KUKA KRL program: f1_Kuka_APT226T02S26.SRC

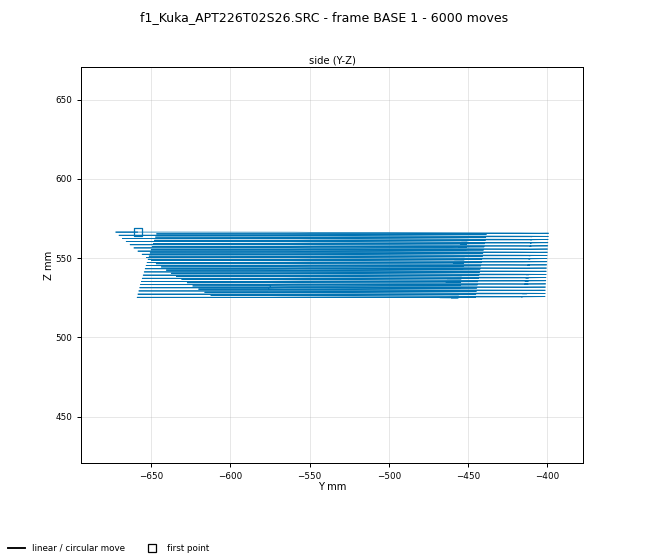
[picture p0: tool path of f1_Kuka_APT226T02S26.SRC in frame BASE 1, 6000 of 6001 moves have a stored position in this frame; points joined in program order, loops and branches not executed]
&ACCESS RVP
&REL 2
&PARAM TEMPLATE = C:\KRC\Roboter\Template\vorgabe
&PARAM EDITMASK = *
DEF f1_Kuka_APT226T02S26()


;FOLD INI;%{PE}%V3.2.0,%MKUKATPBASIS,%CINIT,%VCOMMON,%P
  ;FOLD BAS INI;%{E}%V3.2.0,%MKUKATPBASIS,%CINIT,%VINIT,%P
    GLOBAL INTERRUPT DECL 3 WHEN $STOPMESS==TRUE DO IR_STOPM ( )
    INTERRUPT ON 3
    BAS (#INITMOV,0 )
  ;ENDFOLD (BAS INI)
  ;FOLD USER INI;%{E}%V3.2.0,%MKUKATPUSER,%CINIT,%VINIT,%P
    ;Make your modifications here
  ;ENDFOLD (USER INI)
;ENDFOLD (INI)


;*** Make Null PTP Move
  PTP $pos_act

;*** Auto Load The Correct TOOL Data
  $tool=tool_data[2]

;*** Auto Load The Correct BASE Data
  $base=base_data[1]

  $ADVANCE = 5

;*** Restate Last Velocity
MMPM(30000.0)
SetRPM(8000)
LIN {X 0.091,Y -658.502,Z 566.466,A 0.000,B 0.000,C 90.000,E1 299.922} C_DIS
LIN {X -0.120,Y -661.478,Z 566.462,A 0.000,B 0.000,C 90.000,E1 299.205} C_DIS
LIN {X -0.014,Y -665.940,Z 566.455,A 0.000,B 0.000,C 90.000,E1 297.975} C_DIS
LIN {X 0.167,Y -670.191,Z 566.449,A 0.000,B 0.000,C 90.000,E1 296.744} C_DIS
LIN {X 0.331,Y -670.998,Z 566.447,A 0.000,B 0.000,C 90.000,E1 296.488} C_DIS
LIN {X -0.104,Y -671.526,Z 566.446,A 0.000,B 0.000,C 90.000,E1 296.283} C_DIS
LIN {X -0.059,Y -672.331,Z 566.443,A 0.000,B 0.000,C 90.000,E1 295.796} C_DIS
LIN {X 0.114,Y -672.304,Z 566.442,A 0.000,B 0.000,C 90.000,E1 295.540} C_DIS
LIN {X -0.062,Y -670.081,Z 566.439,A 0.000,B 0.000,C 90.000,E1 294.951} C_DIS
LIN {X 0.021,Y -669.231,Z 566.438,A 0.000,B 0.000,C 90.000,E1 294.823} C_DIS
LIN {X 0.012,Y -665.696,Z 566.436,A 0.000,B 0.000,C 90.000,E1 294.463} C_DIS
LIN {X 0.118,Y -664.657,Z 566.435,A 0.000,B 0.000,C 90.000,E1 294.335} C_DIS
LIN {X 0.191,Y -662.920,Z 566.435,A 0.000,B 0.000,C 90.000,E1 294.207} C_DIS
LIN {X 0.263,Y -660.007,Z 566.434,A 0.000,B 0.000,C 90.000,E1 294.079} C_DIS
LIN {X 0.068,Y -658.610,Z 566.434,A 0.000,B 0.000,C 90.000,E1 294.027} C_DIS
LIN {X -0.130,Y -655.979,Z 566.433,A 0.000,B 0.000,C 90.000,E1 293.875} C_DIS
LIN {X -0.015,Y -649.603,Z 566.431,A 0.000,B 0.000,C 90.000,E1 293.643} C_DIS
LIN {X 0.286,Y -641.955,Z 566.430,A 0.000,B 0.000,C 90.000,E1 293.387} C_DIS
LIN {X -0.348,Y -620.640,Z 566.427,A 0.000,B 0.000,C 90.000,E1 292.898} C_DIS
LIN {X -0.049,Y -600.076,Z 566.424,A 0.000,B 0.000,C 90.000,E1 292.280} C_DIS
LIN {X 0.146,Y -579.548,Z 566.420,A 0.000,B 0.000,C 90.000,E1 291.589} C_DIS
LIN {X 0.178,Y -573.656,Z 566.419,A 0.000,B 0.000,C 90.000,E1 291.354} C_DIS
LIN {X -0.202,Y -567.890,Z 566.417,A 0.000,B 0.000,C 90.000,E1 291.099} C_DIS
LIN {X -0.108,Y -565.511,Z 566.416,A 0.000,B 0.000,C 90.000,E1 290.865} C_DIS
LIN {X 0.054,Y -565.493,Z 566.416,A 0.000,B 0.000,C 90.000,E1 290.844} C_DIS
LIN {X 0.105,Y -565.002,Z 566.415,A 0.000,B 0.000,C 90.000,E1 290.684} C_DIS
LIN {X 0.153,Y -564.693,Z 566.412,A 0.000,B 0.000,C 90.000,E1 290.174} C_DIS
LIN {X 0.335,Y -564.687,Z 566.405,A 0.000,B 0.000,C 90.000,E1 288.779} C_DIS
LIN {X 0.195,Y -564.535,Z 566.398,A 0.000,B 0.000,C 90.000,E1 287.692} C_DIS
LIN {X 0.198,Y -563.994,Z 566.391,A 0.000,B 0.000,C 90.000,E1 286.315} C_DIS
LIN {X 0.039,Y -563.325,Z 566.383,A 0.000,B 0.000,C 90.000,E1 284.954} C_DIS
LIN {X -0.129,Y -562.530,Z 566.375,A 0.000,B 0.000,C 90.000,E1 283.592} C_DIS
LIN {X 0.109,Y -561.743,Z 566.368,A 0.000,B 0.000,C 90.000,E1 282.187} C_DIS
LIN {X -0.215,Y -560.912,Z 566.360,A 0.000,B 0.000,C 90.000,E1 280.838} C_DIS
LIN {X 0.043,Y -559.953,Z 566.351,A 0.000,B 0.000,C 90.000,E1 279.151} C_DIS
LIN {X 0.196,Y -559.248,Z 566.342,A 0.000,B 0.000,C 90.000,E1 277.473} C_DIS
LIN {X -0.153,Y -558.425,Z 566.331,A 0.000,B 0.000,C 90.000,E1 275.568} C_DIS
LIN {X -0.030,Y -557.689,Z 566.320,A 0.000,B 0.000,C 90.000,E1 273.612} C_DIS
LIN {X -0.072,Y -557.116,Z 566.311,A 0.000,B 0.000,C 90.000,E1 271.949} C_DIS
LIN {X -0.206,Y -556.541,Z 566.303,A 0.000,B 0.000,C 90.000,E1 270.573} C_DIS
LIN {X 0.192,Y -555.927,Z 566.295,A 0.000,B 0.000,C 90.000,E1 269.141} C_DIS
LIN {X 0.034,Y -555.274,Z 566.288,A 0.000,B 0.000,C 90.000,E1 267.764} C_DIS
LIN {X -0.133,Y -554.590,Z 566.280,A 0.000,B 0.000,C 90.000,E1 266.388} C_DIS
LIN {X 0.275,Y -553.831,Z 566.272,A 0.000,B 0.000,C 90.000,E1 264.951} C_DIS
LIN {X 0.112,Y -552.989,Z 566.264,A 0.000,B 0.000,C 90.000,E1 263.571} C_DIS
LIN {X -0.049,Y -552.230,Z 566.258,A 0.000,B 0.000,C 90.000,E1 262.470} C_DIS
LIN {X -0.293,Y -551.234,Z 566.252,A 0.000,B 0.000,C 90.000,E1 261.376} C_DIS
LIN {X 0.175,Y -549.737,Z 566.244,A 0.000,B 0.000,C 90.000,E1 259.926} C_DIS
LIN {X -0.258,Y -547.945,Z 566.235,A 0.000,B 0.000,C 90.000,E1 258.285} C_DIS
LIN {X -0.189,Y -546.203,Z 566.225,A 0.000,B 0.000,C 90.000,E1 256.589} C_DIS
LIN {X 0.097,Y -544.289,Z 566.216,A 0.000,B 0.000,C 90.000,E1 254.866} C_DIS
LIN {X 0.116,Y -542.524,Z 566.208,A 0.000,B 0.000,C 90.000,E1 253.449} C_DIS
LIN {X -0.050,Y -540.070,Z 566.199,A 0.000,B 0.000,C 90.000,E1 251.764} C_DIS
LIN {X 0.156,Y -538.266,Z 566.192,A 0.000,B 0.000,C 90.000,E1 250.604} C_DIS
LIN {X -0.135,Y -535.834,Z 566.184,A 0.000,B 0.000,C 90.000,E1 249.209} C_DIS
LIN {X -0.084,Y -532.469,Z 566.175,A 0.000,B 0.000,C 90.000,E1 247.486} C_DIS
LIN {X 0.091,Y -528.786,Z 566.165,A 0.000,B 0.000,C 90.000,E1 245.741} C_DIS
LIN {X 0.230,Y -525.501,Z 566.157,A 0.000,B 0.000,C 90.000,E1 244.280} C_DIS
LIN {X -0.159,Y -521.989,Z 566.149,A 0.000,B 0.000,C 90.000,E1 242.871} C_DIS
LIN {X -0.037,Y -519.122,Z 566.143,A 0.000,B 0.000,C 90.000,E1 241.691} C_DIS
LIN {X 0.046,Y -516.137,Z 566.136,A 0.000,B 0.000,C 90.000,E1 240.511} C_DIS
LIN {X 0.081,Y -512.831,Z 566.130,A 0.000,B 0.000,C 90.000,E1 239.331} C_DIS
LIN {X 0.187,Y -506.734,Z 566.118,A 0.000,B 0.000,C 90.000,E1 237.248} C_DIS
LIN {X -0.020,Y -500.752,Z 566.107,A 0.000,B 0.000,C 90.000,E1 235.182} C_DIS
LIN {X -0.083,Y -493.288,Z 566.092,A 0.000,B 0.000,C 90.000,E1 232.477} C_DIS
LIN {X 0.016,Y -489.998,Z 566.085,A 0.000,B 0.000,C 90.000,E1 231.251} C_DIS
LIN {X -0.175,Y -486.063,Z 566.076,A 0.000,B 0.000,C 90.000,E1 229.747} C_DIS
LIN {X 0.182,Y -480.596,Z 566.064,A 0.000,B 0.000,C 90.000,E1 227.553} C_DIS
LIN {X 0.112,Y -474.437,Z 566.051,A 0.000,B 0.000,C 90.000,E1 225.081} C_DIS
LIN {X -0.068,Y -470.785,Z 566.042,A 0.000,B 0.000,C 90.000,E1 223.542} C_DIS
LIN {X 0.014,Y -467.149,Z 566.033,A 0.000,B 0.000,C 90.000,E1 221.962} C_DIS
LIN {X -0.188,Y -462.845,Z 566.023,A 0.000,B 0.000,C 90.000,E1 220.092} C_DIS
LIN {X -0.252,Y -460.148,Z 566.016,A 0.000,B 0.000,C 90.000,E1 218.830} C_DIS
LIN {X 0.107,Y -455.982,Z 566.005,A 0.000,B 0.000,C 90.000,E1 216.870} C_DIS
LIN {X -0.258,Y -452.625,Z 565.996,A 0.000,B 0.000,C 90.000,E1 215.311} C_DIS
LIN {X -0.238,Y -448.719,Z 565.985,A 0.000,B 0.000,C 90.000,E1 213.372} C_DIS
LIN {X 0.057,Y -444.934,Z 565.974,A 0.000,B 0.000,C 90.000,E1 211.386} C_DIS
LIN {X 0.127,Y -441.936,Z 565.965,A 0.000,B 0.000,C 90.000,E1 209.745} C_DIS
LIN {X 0.041,Y -437.350,Z 565.951,A 0.000,B 0.000,C 90.000,E1 207.129} C_DIS
LIN {X -0.028,Y -433.942,Z 565.940,A 0.000,B 0.000,C 90.000,E1 205.155} C_DIS
LIN {X -0.174,Y -431.214,Z 565.931,A 0.000,B 0.000,C 90.000,E1 203.515} C_DIS
LIN {X 0.020,Y -427.572,Z 565.918,A 0.000,B 0.000,C 90.000,E1 201.153} C_DIS
LIN {X 0.215,Y -425.238,Z 565.908,A 0.000,B 0.000,C 90.000,E1 199.450} C_DIS
LIN {X 0.193,Y -422.028,Z 565.895,A 0.000,B 0.000,C 90.000,E1 197.094} C_DIS
LIN {X -0.161,Y -419.081,Z 565.882,A 0.000,B 0.000,C 90.000,E1 194.773} C_DIS
LIN {X -0.141,Y -417.414,Z 565.874,A 0.000,B 0.000,C 90.000,E1 193.411} C_DIS
LIN {X -0.149,Y -414.490,Z 565.863,A 0.000,B 0.000,C 90.000,E1 191.366} C_DIS
LIN {X -0.153,Y -411.013,Z 565.848,A 0.000,B 0.000,C 90.000,E1 188.624} C_DIS
LIN {X -0.072,Y -408.386,Z 565.834,A 0.000,B 0.000,C 90.000,E1 186.201} C_DIS
LIN {X -0.082,Y -406.582,Z 565.825,A 0.000,B 0.000,C 90.000,E1 184.473} C_DIS
LIN {X 0.071,Y -403.123,Z 565.804,A 0.000,B 0.000,C 90.000,E1 180.630} C_DIS
LIN {X -0.144,Y -401.678,Z 565.792,A 0.000,B 0.000,C 90.000,E1 178.568} C_DIS
LIN {X 0.078,Y -400.698,Z 565.782,A 0.000,B 0.000,C 90.000,E1 176.788} C_DIS
LIN {X 0.151,Y -399.710,Z 565.767,A 0.000,B 0.000,C 90.000,E1 173.976} C_DIS
LIN {X -0.052,Y -399.191,Z 565.749,A 0.000,B 0.000,C 90.000,E1 170.849} C_DIS
LIN {X -0.170,Y -399.159,Z 565.736,A 0.000,B 0.000,C 90.000,E1 168.409} C_DIS
LIN {X 0.025,Y -399.565,Z 565.720,A 0.000,B 0.000,C 90.000,E1 165.574} C_DIS
LIN {X 0.130,Y -399.971,Z 565.712,A 0.000,B 0.000,C 90.000,E1 164.157} C_DIS
LIN {X -0.202,Y -400.926,Z 565.697,A 0.000,B 0.000,C 90.000,E1 161.402} C_DIS
LIN {X 0.084,Y -401.886,Z 565.685,A 0.000,B 0.000,C 90.000,E1 159.263} C_DIS
LIN {X 0.015,Y -402.888,Z 565.673,A 0.000,B 0.000,C 90.000,E1 157.177} C_DIS
LIN {X 0.026,Y -403.897,Z 565.664,A 0.000,B 0.000,C 90.000,E1 155.433} C_DIS
LIN {X 0.112,Y -405.050,Z 565.652,A 0.000,B 0.000,C 90.000,E1 153.332} C_DIS
LIN {X -0.209,Y -406.078,Z 565.642,A 0.000,B 0.000,C 90.000,E1 151.641} C_DIS
LIN {X 0.132,Y -406.794,Z 565.635,A 0.000,B 0.000,C 90.000,E1 150.205} C_DIS
LIN {X 0.039,Y -407.538,Z 565.625,A 0.000,B 0.000,C 90.000,E1 148.486} C_DIS
LIN {X -0.090,Y -408.065,Z 565.617,A 0.000,B 0.000,C 90.000,E1 147.120} C_DIS
LIN {X 0.020,Y -408.430,Z 565.610,A 0.000,B 0.000,C 90.000,E1 145.722} C_DIS
LIN {X 0.053,Y -408.831,Z 565.600,A 0.000,B 0.000,C 90.000,E1 143.989} C_DIS
LIN {X -0.005,Y -409.107,Z 565.590,A 0.000,B 0.000,C 90.000,E1 142.271} C_DIS
LIN {X -0.122,Y -409.308,Z 565.581,A 0.000,B 0.000,C 90.000,E1 140.561} C_DIS
LIN {X -0.083,Y -409.474,Z 565.569,A 0.000,B 0.000,C 90.000,E1 138.485} C_DIS
LIN {X 0.189,Y -409.571,Z 565.558,A 0.000,B 0.000,C 90.000,E1 136.377} C_DIS
LIN {X -0.273,Y -409.836,Z 565.544,A 0.000,B 0.000,C 90.000,E1 134.028} C_DIS
LIN {X -0.141,Y -410.079,Z 565.535,A 0.000,B 0.000,C 90.000,E1 132.285} C_DIS
LIN {X 0.022,Y -410.097,Z 565.525,A 0.000,B 0.000,C 90.000,E1 130.539} C_DIS
LIN {X 0.182,Y -409.998,Z 565.520,A 0.000,B 0.000,C 90.000,E1 129.483} C_DIS
LIN {X 0.080,Y -409.819,Z 565.514,A 0.000,B 0.000,C 90.000,E1 128.463} C_DIS
LIN {X -0.019,Y -409.657,Z 565.511,A 0.000,B 0.000,C 90.000,E1 127.971} C_DIS
LIN {X -0.057,Y -409.666,Z 565.511,A 0.000,B 0.000,C 90.000,E1 127.971} C_DIS
LIN {X -0.188,Y -415.244,Z 565.500,A 0.000,B 0.000,C 90.000,E1 126.091} C_DIS
LIN {X -0.077,Y -416.905,Z 565.497,A 0.000,B 0.000,C 90.000,E1 125.391} C_DIS
LIN {X -0.150,Y -426.632,Z 565.476,A 0.000,B 0.000,C 90.000,E1 121.671} C_DIS
LIN {X -0.187,Y -430.699,Z 565.468,A 0.000,B 0.000,C 90.000,E1 120.335} C_DIS
LIN {X -0.080,Y -437.000,Z 565.454,A 0.000,B 0.000,C 90.000,E1 117.692} C_DIS
LIN {X 0.267,Y -437.037,Z 565.454,A 0.000,B 0.000,C 90.000,E1 117.641} C_DIS
LIN {X -0.240,Y -449.597,Z 565.451,A 0.000,B 0.000,C 90.000,E1 117.129} C_DIS
LIN {X 0.099,Y -461.731,Z 565.448,A 0.000,B 0.000,C 90.000,E1 116.539} C_DIS
LIN {X 0.166,Y -473.663,Z 565.444,A 0.000,B 0.000,C 90.000,E1 115.976} C_DIS
LIN {X -0.213,Y -485.709,Z 565.441,A 0.000,B 0.000,C 90.000,E1 115.463} C_DIS
LIN {X -0.080,Y -495.644,Z 565.439,A 0.000,B 0.000,C 90.000,E1 114.951} C_DIS
LIN {X 0.082,Y -502.219,Z 565.437,A 0.000,B 0.000,C 90.000,E1 114.591} C_DIS
LIN {X 0.151,Y -513.798,Z 565.433,A 0.000,B 0.000,C 90.000,E1 113.951} C_DIS
LIN {X -0.201,Y -525.107,Z 565.430,A 0.000,B 0.000,C 90.000,E1 113.334} C_DIS
LIN {X -0.007,Y -532.885,Z 565.427,A 0.000,B 0.000,C 90.000,E1 112.823} C_DIS
LIN {X 0.033,Y -537.524,Z 565.425,A 0.000,B 0.000,C 90.000,E1 112.514} C_DIS
LIN {X 0.130,Y -546.082,Z 565.422,A 0.000,B 0.000,C 90.000,E1 111.897} C_DIS
LIN {X 0.201,Y -553.885,Z 565.418,A 0.000,B 0.000,C 90.000,E1 111.280} C_DIS
LIN {X 0.052,Y -559.058,Z 565.416,A 0.000,B 0.000,C 90.000,E1 110.844} C_DIS
LIN {X 0.130,Y -563.843,Z 565.413,A 0.000,B 0.000,C 90.000,E1 110.375} C_DIS
LIN {X 0.123,Y -566.067,Z 565.412,A 0.000,B 0.000,C 90.000,E1 110.120} C_DIS
LIN {X 0.206,Y -569.310,Z 565.410,A 0.000,B 0.000,C 90.000,E1 109.758} C_DIS
LIN {X 0.185,Y -573.267,Z 565.407,A 0.000,B 0.000,C 90.000,E1 109.268} C_DIS
LIN {X -0.185,Y -578.969,Z 565.403,A 0.000,B 0.000,C 90.000,E1 108.489} C_DIS
LIN {X -0.093,Y -583.152,Z 565.399,A 0.000,B 0.000,C 90.000,E1 107.819} C_DIS
LIN {X 0.044,Y -589.252,Z 565.393,A 0.000,B 0.000,C 90.000,E1 106.732} C_DIS
LIN {X 0.169,Y -594.082,Z 565.388,A 0.000,B 0.000,C 90.000,E1 105.788} C_DIS
LIN {X 0.006,Y -597.910,Z 565.383,A 0.000,B 0.000,C 90.000,E1 105.009} C_DIS
LIN {X -0.060,Y -600.834,Z 565.380,A 0.000,B 0.000,C 90.000,E1 104.356} C_DIS
LIN {X -0.272,Y -606.577,Z 565.372,A 0.000,B 0.000,C 90.000,E1 103.063} C_DIS
LIN {X -0.133,Y -610.900,Z 565.367,A 0.000,B 0.000,C 90.000,E1 102.007} C_DIS
LIN {X -0.182,Y -615.984,Z 565.359,A 0.000,B 0.000,C 90.000,E1 100.715} C_DIS
LIN {X 0.164,Y -623.736,Z 565.348,A 0.000,B 0.000,C 90.000,E1 98.624} C_DIS
LIN {X -0.289,Y -627.540,Z 565.342,A 0.000,B 0.000,C 90.000,E1 97.644} C_DIS
LIN {X -0.277,Y -632.016,Z 565.335,A 0.000,B 0.000,C 90.000,E1 96.372} C_DIS
LIN {X 0.215,Y -634.479,Z 565.331,A 0.000,B 0.000,C 90.000,E1 95.568} C_DIS
LIN {X 0.108,Y -636.805,Z 565.327,A 0.000,B 0.000,C 90.000,E1 94.821} C_DIS
LIN {X 0.025,Y -638.887,Z 565.323,A 0.000,B 0.000,C 90.000,E1 94.073} C_DIS
LIN {X -0.248,Y -641.332,Z 565.317,A 0.000,B 0.000,C 90.000,E1 93.094} C_DIS
LIN {X 0.081,Y -643.287,Z 565.312,A 0.000,B 0.000,C 90.000,E1 92.064} C_DIS
LIN {X 0.279,Y -644.128,Z 565.309,A 0.000,B 0.000,C 90.000,E1 91.547} C_DIS
LIN {X 0.010,Y -645.490,Z 565.303,A 0.000,B 0.000,C 90.000,E1 90.573} C_DIS
LIN {X -0.016,Y -646.171,Z 565.299,A 0.000,B 0.000,C 90.000,E1 89.828} C_DIS
LIN {X 0.185,Y -646.428,Z 565.296,A 0.000,B 0.000,C 90.000,E1 89.312} C_DIS
LIN {X 0.166,Y -646.585,Z 565.292,A 0.000,B 0.000,C 90.000,E1 88.568} C_DIS
LIN {X 0.166,Y -646.505,Z 565.288,A 0.000,B 0.000,C 90.000,E1 87.822} C_DIS
LIN {X 0.141,Y -646.135,Z 565.284,A 0.000,B 0.000,C 90.000,E1 87.078} C_DIS
LIN {X -0.086,Y -645.321,Z 565.278,A 0.000,B 0.000,C 90.000,E1 86.102} C_DIS
LIN {X -0.273,Y -644.089,Z 565.273,A 0.000,B 0.000,C 90.000,E1 85.122} C_DIS
LIN {X -0.287,Y -643.007,Z 565.269,A 0.000,B 0.000,C 90.000,E1 84.375} C_DIS
LIN {X 0.145,Y -641.255,Z 565.263,A 0.000,B 0.000,C 90.000,E1 83.337} C_DIS
LIN {X -0.350,Y -638.424,Z 565.256,A 0.000,B 0.000,C 90.000,E1 82.129} C_DIS
LIN {X 0.096,Y -635.794,Z 565.251,A 0.000,B 0.000,C 90.000,E1 81.084} C_DIS
LIN {X 0.321,Y -632.160,Z 565.244,A 0.000,B 0.000,C 90.000,E1 79.803} C_DIS
LIN {X -0.135,Y -628.086,Z 565.237,A 0.000,B 0.000,C 90.000,E1 78.578} C_DIS
LIN {X -0.116,Y -625.394,Z 565.232,A 0.000,B 0.000,C 90.000,E1 77.813} C_DIS
LIN {X -0.260,Y -622.564,Z 565.228,A 0.000,B 0.000,C 90.000,E1 77.061} C_DIS
LIN {X 0.228,Y -618.259,Z 565.222,A 0.000,B 0.000,C 90.000,E1 75.992} C_DIS
LIN {X 0.106,Y -614.146,Z 565.217,A 0.000,B 0.000,C 90.000,E1 75.102} C_DIS
LIN {X -0.025,Y -610.337,Z 565.213,A 0.000,B 0.000,C 90.000,E1 74.338} C_DIS
LIN {X 0.010,Y -606.903,Z 565.209,A 0.000,B 0.000,C 90.000,E1 73.685} C_DIS
LIN {X 0.188,Y -603.246,Z 565.206,A 0.000,B 0.000,C 90.000,E1 73.015} C_DIS
LIN {X 0.211,Y -600.152,Z 565.203,A 0.000,B 0.000,C 90.000,E1 72.489} C_DIS
LIN {X -0.232,Y -595.965,Z 565.199,A 0.000,B 0.000,C 90.000,E1 71.873} C_DIS
LIN {X -0.079,Y -592.202,Z 565.196,A 0.000,B 0.000,C 90.000,E1 71.329} C_DIS
LIN {X 0.274,Y -586.514,Z 565.192,A 0.000,B 0.000,C 90.000,E1 70.550} C_DIS
LIN {X -0.192,Y -581.956,Z 565.189,A 0.000,B 0.000,C 90.000,E1 70.061} C_DIS
LIN {X -0.114,Y -577.144,Z 565.186,A 0.000,B 0.000,C 90.000,E1 69.518} C_DIS
LIN {X 0.224,Y -571.989,Z 565.183,A 0.000,B 0.000,C 90.000,E1 68.954} C_DIS
LIN {X -0.098,Y -569.075,Z 565.182,A 0.000,B 0.000,C 90.000,E1 68.720} C_DIS
LIN {X -0.122,Y -567.051,Z 565.181,A 0.000,B 0.000,C 90.000,E1 68.518} C_DIS
LIN {X 0.117,Y -563.879,Z 565.179,A 0.000,B 0.000,C 90.000,E1 68.230} C_DIS
LIN {X 0.190,Y -561.737,Z 565.178,A 0.000,B 0.000,C 90.000,E1 68.028} C_DIS
LIN {X 0.310,Y -555.590,Z 565.175,A 0.000,B 0.000,C 90.000,E1 67.539} C_DIS
LIN {X -0.179,Y -549.616,Z 565.173,A 0.000,B 0.000,C 90.000,E1 67.177} C_DIS
LIN {X 0.018,Y -544.631,Z 565.171,A 0.000,B 0.000,C 90.000,E1 66.847} C_DIS
LIN {X 0.166,Y -538.455,Z 565.169,A 0.000,B 0.000,C 90.000,E1 66.485} C_DIS
LIN {X -0.132,Y -531.737,Z 565.168,A 0.000,B 0.000,C 90.000,E1 66.177} C_DIS
LIN {X -0.018,Y -528.225,Z 565.167,A 0.000,B 0.000,C 90.000,E1 65.997} C_DIS
LIN {X -0.065,Y -516.079,Z 565.164,A 0.000,B 0.000,C 90.000,E1 65.485} C_DIS
LIN {X -0.140,Y -507.333,Z 565.162,A 0.000,B 0.000,C 90.000,E1 65.153} C_DIS
LIN {X -0.033,Y -482.787,Z 565.157,A 0.000,B 0.000,C 90.000,E1 64.229} C_DIS
LIN {X 0.134,Y -463.845,Z 565.153,A 0.000,B 0.000,C 90.000,E1 63.461} C_DIS
LIN {X -0.021,Y -457.694,Z 565.151,A 0.000,B 0.000,C 90.000,E1 63.204} C_DIS
LIN {X -0.056,Y -457.648,Z 565.151,A 0.000,B 0.000,C 90.000,E1 63.204} C_DIS
LIN {X -0.008,Y -455.803,Z 565.145,A 0.000,B 0.000,C 90.000,E1 62.103} C_DIS
LIN {X 0.096,Y -455.205,Z 565.143,A 0.000,B 0.000,C 90.000,E1 61.769} C_DIS
LIN {X -0.056,Y -446.529,Z 565.122,A 0.000,B 0.000,C 90.000,E1 57.916} C_DIS
LIN {X -0.165,Y -444.146,Z 565.115,A 0.000,B 0.000,C 90.000,E1 56.628} C_DIS
LIN {X -0.053,Y -442.565,Z 565.111,A 0.000,B 0.000,C 90.000,E1 55.960} C_DIS
LIN {X 0.165,Y -438.365,Z 565.101,A 0.000,B 0.000,C 90.000,E1 54.196} C_DIS
LIN {X 0.125,Y -438.357,Z 565.101,A 0.000,B 0.000,C 90.000,E1 54.196} C_DIS
LIN {X -0.110,Y -441.521,Z 565.087,A 0.000,B 0.000,C 90.000,E1 51.698} C_DIS
LIN {X -0.174,Y -442.811,Z 565.082,A 0.000,B 0.000,C 90.000,E1 50.723} C_DIS
LIN {X -0.249,Y -445.229,Z 565.071,A 0.000,B 0.000,C 90.000,E1 48.771} C_DIS
LIN {X 0.031,Y -447.166,Z 565.062,A 0.000,B 0.000,C 90.000,E1 47.106} C_DIS
LIN {X 0.000,Y -448.679,Z 565.055,A 0.000,B 0.000,C 90.000,E1 45.810} C_DIS
LIN {X -0.003,Y -449.663,Z 565.049,A 0.000,B 0.000,C 90.000,E1 44.838} C_DIS
LIN {X 0.010,Y -450.802,Z 565.042,A 0.000,B 0.000,C 90.000,E1 43.542} C_DIS
LIN {X 0.058,Y -451.689,Z 565.035,A 0.000,B 0.000,C 90.000,E1 42.243} C_DIS
LIN {X 0.133,Y -452.421,Z 565.026,A 0.000,B 0.000,C 90.000,E1 40.620} C_DIS
LIN {X -0.085,Y -452.674,Z 565.019,A 0.000,B 0.000,C 90.000,E1 39.358} C_DIS
LIN {X -0.016,Y -452.799,Z 565.013,A 0.000,B 0.000,C 90.000,E1 38.382} C_DIS
LIN {X 0.122,Y -452.730,Z 565.006,A 0.000,B 0.000,C 90.000,E1 37.076} C_DIS
LIN {X 0.072,Y -452.492,Z 564.997,A 0.000,B 0.000,C 90.000,E1 35.471} C_DIS
LIN {X 0.074,Y -451.782,Z 564.985,A 0.000,B 0.000,C 90.000,E1 33.214} C_DIS
LIN {X 0.219,Y -451.328,Z 564.974,A 0.000,B 0.000,C 90.000,E1 31.258} C_DIS
LIN {X 0.036,Y -451.029,Z 564.965,A 0.000,B 0.000,C 90.000,E1 29.667} C_DIS
LIN {X 0.191,Y -450.546,Z 564.952,A 0.000,B 0.000,C 90.000,E1 27.385} C_DIS
LIN {X -0.028,Y -450.178,Z 564.943,A 0.000,B 0.000,C 90.000,E1 25.796} C_DIS
LIN {X -0.252,Y -449.954,Z 564.934,A 0.000,B 0.000,C 90.000,E1 24.207} C_DIS
LIN {X 0.094,Y -449.708,Z 564.922,A 0.000,B 0.000,C 90.000,E1 21.897} C_DIS
LIN {X 0.095,Y -449.600,Z 564.909,A 0.000,B 0.000,C 90.000,E1 19.631} C_DIS
LIN {X -0.202,Y -449.669,Z 564.897,A 0.000,B 0.000,C 90.000,E1 17.402} C_DIS
LIN {X 0.107,Y -450.046,Z 564.882,A 0.000,B 0.000,C 90.000,E1 14.773} C_DIS
LIN {X -0.103,Y -450.683,Z 564.870,A 0.000,B 0.000,C 90.000,E1 12.535} C_DIS
LIN {X 0.050,Y -451.603,Z 564.857,A 0.000,B 0.000,C 90.000,E1 10.254} C_DIS
LIN {X 0.175,Y -452.471,Z 564.848,A 0.000,B 0.000,C 90.000,E1 8.624} C_DIS
LIN {X -0.141,Y -454.065,Z 564.834,A 0.000,B 0.000,C 90.000,E1 6.087} C_DIS
LIN {X 0.082,Y -455.571,Z 564.823,A 0.000,B 0.000,C 90.000,E1 4.131} C_DIS
LIN {X -0.219,Y -457.811,Z 564.809,A 0.000,B 0.000,C 90.000,E1 1.604} C_DIS
LIN {X -0.147,Y -460.823,Z 564.794,A 0.000,B 0.000,C 90.000,E1 358.854} C_DIS
LIN {X 0.159,Y -464.118,Z 564.779,A 0.000,B 0.000,C 90.000,E1 356.274} C_DIS
LIN {X 0.159,Y -466.798,Z 564.769,A 0.000,B 0.000,C 90.000,E1 354.375} C_DIS
LIN {X 0.000,Y -469.127,Z 564.760,A 0.000,B 0.000,C 90.000,E1 352.818} C_DIS
LIN {X -0.054,Y -471.385,Z 564.751,A 0.000,B 0.000,C 90.000,E1 351.254} C_DIS
LIN {X -0.238,Y -474.139,Z 564.741,A 0.000,B 0.000,C 90.000,E1 349.398} C_DIS
LIN {X -0.026,Y -476.585,Z 564.732,A 0.000,B 0.000,C 90.000,E1 347.813} C_DIS
LIN {X -0.094,Y -480.574,Z 564.719,A 0.000,B 0.000,C 90.000,E1 345.338} C_DIS
LIN {X 0.067,Y -485.614,Z 564.703,A 0.000,B 0.000,C 90.000,E1 342.543} C_DIS
LIN {X -0.163,Y -489.177,Z 564.693,A 0.000,B 0.000,C 90.000,E1 340.732} C_DIS
LIN {X -0.188,Y -492.149,Z 564.684,A 0.000,B 0.000,C 90.000,E1 339.209} C_DIS
LIN {X -0.027,Y -494.423,Z 564.678,A 0.000,B 0.000,C 90.000,E1 337.975} C_DIS
LIN {X -0.236,Y -497.287,Z 564.669,A 0.000,B 0.000,C 90.000,E1 336.485} C_DIS
LIN {X -0.192,Y -499.962,Z 564.661,A 0.000,B 0.000,C 90.000,E1 334.973} C_DIS
LIN {X -0.104,Y -502.524,Z 564.653,A 0.000,B 0.000,C 90.000,E1 333.461} C_DIS
LIN {X 0.179,Y -504.561,Z 564.646,A 0.000,B 0.000,C 90.000,E1 332.231} C_DIS
LIN {X -0.002,Y -507.496,Z 564.636,A 0.000,B 0.000,C 90.000,E1 330.461} C_DIS
LIN {X 0.108,Y -511.464,Z 564.623,A 0.000,B 0.000,C 90.000,E1 328.074} C_DIS
LIN {X 0.170,Y -514.489,Z 564.613,A 0.000,B 0.000,C 90.000,E1 326.294} C_DIS
LIN {X -0.064,Y -517.057,Z 564.605,A 0.000,B 0.000,C 90.000,E1 324.848} C_DIS
LIN {X 0.041,Y -519.683,Z 564.597,A 0.000,B 0.000,C 90.000,E1 323.371} C_DIS
LIN {X -0.045,Y -523.919,Z 564.584,A 0.000,B 0.000,C 90.000,E1 321.045} C_DIS
LIN {X -0.047,Y -528.029,Z 564.572,A 0.000,B 0.000,C 90.000,E1 319.013} C_DIS
LIN {X -0.004,Y -533.253,Z 564.560,A 0.000,B 0.000,C 90.000,E1 316.701} C_DIS
LIN {X -0.177,Y -537.393,Z 564.550,A 0.000,B 0.000,C 90.000,E1 315.000} C_DIS
LIN {X -0.213,Y -538.687,Z 564.547,A 0.000,B 0.000,C 90.000,E1 314.433} C_DIS
LIN {X 0.115,Y -542.821,Z 564.539,A 0.000,B 0.000,C 90.000,E1 312.975} C_DIS
LIN {X -0.161,Y -545.204,Z 564.535,A 0.000,B 0.000,C 90.000,E1 312.366} C_DIS
LIN {X -0.039,Y -547.320,Z 564.533,A 0.000,B 0.000,C 90.000,E1 312.000} C_DIS
LIN {X 0.160,Y -548.035,Z 564.533,A 0.000,B 0.000,C 90.000,E1 311.838} C_DIS
LIN {X -0.214,Y -550.099,Z 564.531,A 0.000,B 0.000,C 90.000,E1 311.595} C_DIS
LIN {X -0.011,Y -550.977,Z 564.530,A 0.000,B 0.000,C 90.000,E1 311.434} C_DIS
LIN {X -0.171,Y -552.096,Z 564.529,A 0.000,B 0.000,C 90.000,E1 311.310} C_DIS
LIN {X 0.012,Y -553.582,Z 564.529,A 0.000,B 0.000,C 90.000,E1 311.148} C_DIS
LIN {X -0.157,Y -555.670,Z 564.527,A 0.000,B 0.000,C 90.000,E1 310.906} C_DIS
LIN {X 0.040,Y -560.191,Z 564.525,A 0.000,B 0.000,C 90.000,E1 310.458} C_DIS
LIN {X -0.289,Y -566.071,Z 564.522,A 0.000,B 0.000,C 90.000,E1 310.011} C_DIS
LIN {X -0.235,Y -576.106,Z 564.518,A 0.000,B 0.000,C 90.000,E1 309.277} C_DIS
LIN {X -0.055,Y -586.453,Z 564.514,A 0.000,B 0.000,C 90.000,E1 308.508} C_DIS
LIN {X -0.329,Y -592.161,Z 564.512,A 0.000,B 0.000,C 90.000,E1 308.096} C_DIS
LIN {X -0.321,Y -598.973,Z 564.508,A 0.000,B 0.000,C 90.000,E1 307.523} C_DIS
LIN {X -0.155,Y -604.172,Z 564.506,A 0.000,B 0.000,C 90.000,E1 307.030} C_DIS
LIN {X -0.165,Y -607.955,Z 564.504,A 0.000,B 0.000,C 90.000,E1 306.664} C_DIS
LIN {X 0.052,Y -612.817,Z 564.501,A 0.000,B 0.000,C 90.000,E1 306.137} C_DIS
LIN {X -0.272,Y -619.839,Z 564.497,A 0.000,B 0.000,C 90.000,E1 305.391} C_DIS
LIN {X 0.174,Y -628.577,Z 564.491,A 0.000,B 0.000,C 90.000,E1 304.326} C_DIS
LIN {X 0.013,Y -634.783,Z 564.487,A 0.000,B 0.000,C 90.000,E1 303.579} C_DIS
LIN {X -0.102,Y -639.721,Z 564.483,A 0.000,B 0.000,C 90.000,E1 302.959} C_DIS
LIN {X -0.182,Y -643.971,Z 564.480,A 0.000,B 0.000,C 90.000,E1 302.339} C_DIS
LIN {X 0.285,Y -647.097,Z 564.477,A 0.000,B 0.000,C 90.000,E1 301.799} C_DIS
LIN {X -0.074,Y -650.468,Z 564.473,A 0.000,B 0.000,C 90.000,E1 301.209} C_DIS
LIN {X 0.025,Y -654.513,Z 564.469,A 0.000,B 0.000,C 90.000,E1 300.335} C_DIS
LIN {X 0.220,Y -658.730,Z 564.463,A 0.000,B 0.000,C 90.000,E1 299.333} C_DIS
LIN {X 0.279,Y -663.216,Z 564.456,A 0.000,B 0.000,C 90.000,E1 298.103} C_DIS
LIN {X -0.177,Y -667.563,Z 564.450,A 0.000,B 0.000,C 90.000,E1 296.924} C_DIS
LIN {X 0.132,Y -669.149,Z 564.447,A 0.000,B 0.000,C 90.000,E1 296.411} C_DIS
LIN {X 0.160,Y -670.059,Z 564.444,A 0.000,B 0.000,C 90.000,E1 295.924} C_DIS
LIN {X -0.279,Y -670.256,Z 564.443,A 0.000,B 0.000,C 90.000,E1 295.720} C_DIS
LIN {X -0.114,Y -669.973,Z 564.441,A 0.000,B 0.000,C 90.000,E1 295.463} C_DIS
LIN {X 0.052,Y -669.123,Z 564.440,A 0.000,B 0.000,C 90.000,E1 295.207} C_DIS
LIN {X 0.215,Y -668.096,Z 564.439,A 0.000,B 0.000,C 90.000,E1 294.951} C_DIS
LIN {X 0.014,Y -667.068,Z 564.438,A 0.000,B 0.000,C 90.000,E1 294.847} C_DIS
LIN {X 0.096,Y -665.847,Z 564.437,A 0.000,B 0.000,C 90.000,E1 294.719} C_DIS
LIN {X -0.295,Y -664.134,Z 564.436,A 0.000,B 0.000,C 90.000,E1 294.515} C_DIS
LIN {X -0.223,Y -662.944,Z 564.435,A 0.000,B 0.000,C 90.000,E1 294.387} C_DIS
LIN {X -0.150,Y -660.945,Z 564.435,A 0.000,B 0.000,C 90.000,E1 294.259} C_DIS
LIN {X -0.004,Y -659.139,Z 564.434,A 0.000,B 0.000,C 90.000,E1 294.155} C_DIS
LIN {X 0.146,Y -656.365,Z 564.433,A 0.000,B 0.000,C 90.000,E1 293.951} C_DIS
LIN {X -0.119,Y -654.664,Z 564.433,A 0.000,B 0.000,C 90.000,E1 293.875} C_DIS
LIN {X -0.096,Y -649.752,Z 564.432,A 0.000,B 0.000,C 90.000,E1 293.695} C_DIS
LIN {X 0.221,Y -640.602,Z 564.430,A 0.000,B 0.000,C 90.000,E1 293.387} C_DIS
LIN {X 0.091,Y -621.538,Z 564.427,A 0.000,B 0.000,C 90.000,E1 292.898} C_DIS
LIN {X -0.170,Y -601.106,Z 564.424,A 0.000,B 0.000,C 90.000,E1 292.333} C_DIS
LIN {X -0.148,Y -580.528,Z 564.420,A 0.000,B 0.000,C 90.000,E1 291.663} C_DIS
LIN {X 0.043,Y -573.386,Z 564.419,A 0.000,B 0.000,C 90.000,E1 291.354} C_DIS
LIN {X 0.224,Y -568.086,Z 564.417,A 0.000,B 0.000,C 90.000,E1 291.046} C_DIS
LIN {X 0.017,Y -566.082,Z 564.416,A 0.000,B 0.000,C 90.000,E1 290.865} C_DIS
LIN {X -0.024,Y -566.046,Z 564.416,A 0.000,B 0.000,C 90.000,E1 290.865} C_DIS
LIN {X 0.193,Y -565.520,Z 564.415,A 0.000,B 0.000,C 90.000,E1 290.663} C_DIS
LIN {X -0.203,Y -565.309,Z 564.413,A 0.000,B 0.000,C 90.000,E1 290.429} C_DIS
LIN {X -0.066,Y -565.165,Z 564.403,A 0.000,B 0.000,C 90.000,E1 288.489} C_DIS
LIN {X -0.194,Y -564.948,Z 564.397,A 0.000,B 0.000,C 90.000,E1 287.402} C_DIS
LIN {X -0.177,Y -564.356,Z 564.389,A 0.000,B 0.000,C 90.000,E1 286.024} C_DIS
LIN {X -0.181,Y -563.658,Z 564.381,A 0.000,B 0.000,C 90.000,E1 284.647} C_DIS
LIN {X 0.066,Y -562.845,Z 564.374,A 0.000,B 0.000,C 90.000,E1 283.244} C_DIS
LIN {X 0.275,Y -562.214,Z 564.368,A 0.000,B 0.000,C 90.000,E1 282.119} C_DIS
LIN {X -0.157,Y -561.407,Z 564.360,A 0.000,B 0.000,C 90.000,E1 280.782} C_DIS
LIN {X 0.114,Y -560.465,Z 564.351,A 0.000,B 0.000,C 90.000,E1 279.095} C_DIS
LIN {X -0.201,Y -559.791,Z 564.341,A 0.000,B 0.000,C 90.000,E1 277.466} C_DIS
LIN {X -0.054,Y -558.936,Z 564.331,A 0.000,B 0.000,C 90.000,E1 275.511} C_DIS
LIN {X 0.084,Y -558.205,Z 564.320,A 0.000,B 0.000,C 90.000,E1 273.555} C_DIS
LIN {X 0.054,Y -557.602,Z 564.311,A 0.000,B 0.000,C 90.000,E1 271.892} C_DIS
LIN {X -0.073,Y -557.024,Z 564.303,A 0.000,B 0.000,C 90.000,E1 270.516} C_DIS
LIN {X -0.223,Y -556.402,Z 564.295,A 0.000,B 0.000,C 90.000,E1 269.141} C_DIS
LIN {X 0.260,Y -555.547,Z 564.286,A 0.000,B 0.000,C 90.000,E1 267.421} C_DIS
LIN {X 0.023,Y -555.000,Z 564.280,A 0.000,B 0.000,C 90.000,E1 266.331} C_DIS
LIN {X -0.224,Y -554.397,Z 564.273,A 0.000,B 0.000,C 90.000,E1 265.241} C_DIS
LIN {X -0.270,Y -553.367,Z 564.264,A 0.000,B 0.000,C 90.000,E1 263.571} C_DIS
LIN {X 0.164,Y -552.396,Z 564.256,A 0.000,B 0.000,C 90.000,E1 262.129} C_DIS
LIN {X -0.118,Y -551.618,Z 564.252,A 0.000,B 0.000,C 90.000,E1 261.319} C_DIS
LIN {X -0.187,Y -550.118,Z 564.244,A 0.000,B 0.000,C 90.000,E1 259.926} C_DIS
LIN {X -0.181,Y -548.577,Z 564.236,A 0.000,B 0.000,C 90.000,E1 258.522} C_DIS
LIN {X -0.100,Y -546.858,Z 564.227,A 0.000,B 0.000,C 90.000,E1 256.825} C_DIS
LIN {X 0.199,Y -544.907,Z 564.217,A 0.000,B 0.000,C 90.000,E1 255.102} C_DIS
LIN {X -0.060,Y -542.797,Z 564.208,A 0.000,B 0.000,C 90.000,E1 253.433} C_DIS
LIN {X 0.139,Y -540.271,Z 564.199,A 0.000,B 0.000,C 90.000,E1 251.710} C_DIS
LIN {X 0.123,Y -538.899,Z 564.194,A 0.000,B 0.000,C 90.000,E1 250.859} C_DIS
LIN {X 0.026,Y -536.476,Z 564.186,A 0.000,B 0.000,C 90.000,E1 249.444} C_DIS
LIN {X -0.026,Y -534.844,Z 564.181,A 0.000,B 0.000,C 90.000,E1 248.592} C_DIS
LIN {X 0.096,Y -532.588,Z 564.175,A 0.000,B 0.000,C 90.000,E1 247.433} C_DIS
LIN {X 0.082,Y -529.484,Z 564.167,A 0.000,B 0.000,C 90.000,E1 245.997} C_DIS
LIN {X -0.074,Y -525.552,Z 564.157,A 0.000,B 0.000,C 90.000,E1 244.280} C_DIS
LIN {X 0.005,Y -521.984,Z 564.149,A 0.000,B 0.000,C 90.000,E1 242.820} C_DIS
LIN {X -0.208,Y -518.373,Z 564.141,A 0.000,B 0.000,C 90.000,E1 241.385} C_DIS
LIN {X 0.198,Y -516.122,Z 564.136,A 0.000,B 0.000,C 90.000,E1 240.461} C_DIS
LIN {X -0.127,Y -513.684,Z 564.131,A 0.000,B 0.000,C 90.000,E1 239.616} C_DIS
LIN {X -0.066,Y -508.391,Z 564.121,A 0.000,B 0.000,C 90.000,E1 237.837} C_DIS
LIN {X 0.313,Y -503.196,Z 564.111,A 0.000,B 0.000,C 90.000,E1 236.008} C_DIS
LIN {X -0.143,Y -498.940,Z 564.103,A 0.000,B 0.000,C 90.000,E1 234.562} C_DIS
LIN {X 0.017,Y -493.169,Z 564.091,A 0.000,B 0.000,C 90.000,E1 232.431} C_DIS
LIN {X 0.242,Y -487.522,Z 564.080,A 0.000,B 0.000,C 90.000,E1 230.275} C_DIS
LIN {X -0.177,Y -482.779,Z 564.069,A 0.000,B 0.000,C 90.000,E1 228.485} C_DIS
LIN {X -0.109,Y -480.476,Z 564.064,A 0.000,B 0.000,C 90.000,E1 227.553} C_DIS
LIN {X -0.179,Y -474.317,Z 564.050,A 0.000,B 0.000,C 90.000,E1 225.081} C_DIS
LIN {X -0.018,Y -470.670,Z 564.042,A 0.000,B 0.000,C 90.000,E1 223.500} C_DIS
LIN {X 0.071,Y -467.013,Z 564.033,A 0.000,B 0.000,C 90.000,E1 221.919} C_DIS
LIN {X 0.122,Y -463.448,Z 564.024,A 0.000,B 0.000,C 90.000,E1 220.334} C_DIS
LIN {X 0.103,Y -460.005,Z 564.015,A 0.000,B 0.000,C 90.000,E1 218.749} C_DIS
LIN {X -0.184,Y -455.842,Z 564.005,A 0.000,B 0.000,C 90.000,E1 216.870} C_DIS
LIN {X 0.168,Y -451.824,Z 563.994,A 0.000,B 0.000,C 90.000,E1 214.898} C_DIS
LIN {X -0.134,Y -447.256,Z 563.981,A 0.000,B 0.000,C 90.000,E1 212.673} C_DIS
LIN {X 0.143,Y -444.766,Z 563.974,A 0.000,B 0.000,C 90.000,E1 211.337} C_DIS
LIN {X -0.118,Y -441.186,Z 563.963,A 0.000,B 0.000,C 90.000,E1 209.411} C_DIS
LIN {X 0.133,Y -437.175,Z 563.951,A 0.000,B 0.000,C 90.000,E1 207.078} C_DIS
LIN {X 0.065,Y -433.780,Z 563.940,A 0.000,B 0.000,C 90.000,E1 205.103} C_DIS
LIN {X -0.079,Y -431.048,Z 563.930,A 0.000,B 0.000,C 90.000,E1 203.462} C_DIS
LIN {X -0.087,Y -427.942,Z 563.919,A 0.000,B 0.000,C 90.000,E1 201.461} C_DIS
LIN {X -0.088,Y -425.088,Z 563.908,A 0.000,B 0.000,C 90.000,E1 199.450} C_DIS
LIN {X 0.111,Y -422.376,Z 563.897,A 0.000,B 0.000,C 90.000,E1 197.402} C_DIS
LIN {X -0.060,Y -418.993,Z 563.882,A 0.000,B 0.000,C 90.000,E1 194.717} C_DIS
LIN {X -0.095,Y -417.803,Z 563.876,A 0.000,B 0.000,C 90.000,E1 193.703} C_DIS
LIN {X 0.159,Y -416.324,Z 563.870,A 0.000,B 0.000,C 90.000,E1 192.647} C_DIS
LIN {X -0.158,Y -412.215,Z 563.853,A 0.000,B 0.000,C 90.000,E1 189.613} C_DIS
LIN {X 0.056,Y -408.721,Z 563.836,A 0.000,B 0.000,C 90.000,E1 186.486} C_DIS
LIN {X 0.021,Y -406.566,Z 563.825,A 0.000,B 0.000,C 90.000,E1 184.416} C_DIS
LIN {X -0.196,Y -403.423,Z 563.805,A 0.000,B 0.000,C 90.000,E1 180.974} C_DIS
LIN {X -0.040,Y -401.710,Z 563.792,A 0.000,B 0.000,C 90.000,E1 178.511} C_DIS
LIN {X 0.012,Y -400.178,Z 563.774,A 0.000,B 0.000,C 90.000,E1 175.355} C_DIS
LIN {X -0.177,Y -399.634,Z 563.763,A 0.000,B 0.000,C 90.000,E1 173.280} C_DIS
LIN {X 0.022,Y -399.294,Z 563.745,A 0.000,B 0.000,C 90.000,E1 170.095} C_DIS
LIN {X -0.041,Y -399.406,Z 563.729,A 0.000,B 0.000,C 90.000,E1 167.297} C_DIS
LIN {X -0.149,Y -400.129,Z 563.712,A 0.000,B 0.000,C 90.000,E1 164.157} C_DIS
LIN {X 0.032,Y -401.095,Z 563.696,A 0.000,B 0.000,C 90.000,E1 161.329} C_DIS
LIN {X 0.189,Y -402.052,Z 563.685,A 0.000,B 0.000,C 90.000,E1 159.209} C_DIS
LIN {X 0.079,Y -403.491,Z 563.669,A 0.000,B 0.000,C 90.000,E1 156.433} C_DIS
LIN {X -0.098,Y -404.481,Z 563.659,A 0.000,B 0.000,C 90.000,E1 154.717} C_DIS
LIN {X 0.177,Y -406.125,Z 563.644,A 0.000,B 0.000,C 90.000,E1 151.897} C_DIS
LIN {X -0.122,Y -407.037,Z 563.634,A 0.000,B 0.000,C 90.000,E1 150.205} C_DIS
LIN {X 0.003,Y -407.765,Z 563.625,A 0.000,B 0.000,C 90.000,E1 148.456} C_DIS
LIN {X 0.143,Y -408.378,Z 563.615,A 0.000,B 0.000,C 90.000,E1 146.707} C_DIS
LIN {X 0.114,Y -408.674,Z 563.609,A 0.000,B 0.000,C 90.000,E1 145.674} C_DIS
LIN {X -0.186,Y -409.091,Z 563.600,A 0.000,B 0.000,C 90.000,E1 143.989} C_DIS
LIN {X -0.238,Y -409.364,Z 563.590,A 0.000,B 0.000,C 90.000,E1 142.271} C_DIS
LIN {X -0.035,Y -409.527,Z 563.581,A 0.000,B 0.000,C 90.000,E1 140.517} C_DIS
LIN {X 0.119,Y -409.671,Z 563.571,A 0.000,B 0.000,C 90.000,E1 138.771} C_DIS
LIN {X 0.121,Y -409.747,Z 563.560,A 0.000,B 0.000,C 90.000,E1 136.701} C_DIS
LIN {X 0.242,Y -409.987,Z 563.546,A 0.000,B 0.000,C 90.000,E1 134.271} C_DIS
LIN {X -0.201,Y -410.236,Z 563.537,A 0.000,B 0.000,C 90.000,E1 132.609} C_DIS
LIN {X -0.030,Y -410.301,Z 563.527,A 0.000,B 0.000,C 90.000,E1 130.862} C_DIS
LIN {X 0.136,Y -410.286,Z 563.521,A 0.000,B 0.000,C 90.000,E1 129.806} C_DIS
LIN {X -0.119,Y -410.000,Z 563.514,A 0.000,B 0.000,C 90.000,E1 128.463} C_DIS
LIN {X -0.119,Y -409.793,Z 563.511,A 0.000,B 0.000,C 90.000,E1 127.935} C_DIS
LIN {X 0.165,Y -409.803,Z 563.511,A 0.000,B 0.000,C 90.000,E1 127.890} C_DIS
LIN {X 0.195,Y -415.328,Z 563.500,A 0.000,B 0.000,C 90.000,E1 126.011} C_DIS
LIN {X -0.148,Y -418.583,Z 563.493,A 0.000,B 0.000,C 90.000,E1 124.692} C_DIS
LIN {X 0.212,Y -428.712,Z 563.472,A 0.000,B 0.000,C 90.000,E1 120.924} C_DIS
LIN {X 0.202,Y -430.773,Z 563.468,A 0.000,B 0.000,C 90.000,E1 120.256} C_DIS
LIN {X 0.129,Y -437.732,Z 563.452,A 0.000,B 0.000,C 90.000,E1 117.385} C_DIS
LIN {X 0.089,Y -437.794,Z 563.452,A 0.000,B 0.000,C 90.000,E1 117.385} C_DIS
LIN {X -0.120,Y -460.944,Z 563.446,A 0.000,B 0.000,C 90.000,E1 116.360} C_DIS
LIN {X -0.021,Y -472.889,Z 563.443,A 0.000,B 0.000,C 90.000,E1 115.796} C_DIS
LIN {X 0.291,Y -484.997,Z 563.440,A 0.000,B 0.000,C 90.000,E1 115.207} C_DIS
LIN {X -0.163,Y -494.941,Z 563.438,A 0.000,B 0.000,C 90.000,E1 114.771} C_DIS
LIN {X 0.220,Y -501.677,Z 563.436,A 0.000,B 0.000,C 90.000,E1 114.387} C_DIS
LIN {X 0.040,Y -514.814,Z 563.432,A 0.000,B 0.000,C 90.000,E1 113.695} C_DIS
LIN {X 0.098,Y -524.575,Z 563.429,A 0.000,B 0.000,C 90.000,E1 113.131} C_DIS
LIN {X 0.165,Y -532.372,Z 563.426,A 0.000,B 0.000,C 90.000,E1 112.642} C_DIS
LIN {X -0.113,Y -538.331,Z 563.424,A 0.000,B 0.000,C 90.000,E1 112.280} C_DIS
LIN {X -0.132,Y -541.470,Z 563.423,A 0.000,B 0.000,C 90.000,E1 112.078} C_DIS
LIN {X -0.081,Y -547.464,Z 563.420,A 0.000,B 0.000,C 90.000,E1 111.642} C_DIS
LIN {X 0.081,Y -552.739,Z 563.418,A 0.000,B 0.000,C 90.000,E1 111.227} C_DIS
LIN {X -0.018,Y -558.046,Z 563.416,A 0.000,B 0.000,C 90.000,E1 110.791} C_DIS
LIN {X -0.008,Y -563.246,Z 563.413,A 0.000,B 0.000,C 90.000,E1 110.301} C_DIS
LIN {X 0.100,Y -568.271,Z 563.410,A 0.000,B 0.000,C 90.000,E1 109.758} C_DIS
LIN {X 0.003,Y -573.825,Z 563.406,A 0.000,B 0.000,C 90.000,E1 109.087} C_DIS
LIN {X -0.002,Y -577.707,Z 563.403,A 0.000,B 0.000,C 90.000,E1 108.544} C_DIS
LIN {X 0.086,Y -582.754,Z 563.399,A 0.000,B 0.000,C 90.000,E1 107.764} C_DIS
LIN {X -0.070,Y -588.132,Z 563.394,A 0.000,B 0.000,C 90.000,E1 106.858} C_DIS
LIN {X 0.023,Y -591.098,Z 563.391,A 0.000,B 0.000,C 90.000,E1 106.315} C_DIS
LIN {X -0.101,Y -594.610,Z 563.387,A 0.000,B 0.000,C 90.000,E1 105.662} C_DIS
LIN {X 0.093,Y -599.114,Z 563.382,A 0.000,B 0.000,C 90.000,E1 104.717} C_DIS
LIN {X -0.241,Y -603.269,Z 563.377,A 0.000,B 0.000,C 90.000,E1 103.828} C_DIS
LIN {X -0.146,Y -607.876,Z 563.371,A 0.000,B 0.000,C 90.000,E1 102.771} C_DIS
LIN {X 0.266,Y -611.230,Z 563.367,A 0.000,B 0.000,C 90.000,E1 101.951} C_DIS
LIN {X 0.228,Y -616.370,Z 563.359,A 0.000,B 0.000,C 90.000,E1 100.658} C_DIS
LIN {X -0.339,Y -625.141,Z 563.347,A 0.000,B 0.000,C 90.000,E1 98.398} C_DIS
LIN {X -0.066,Y -628.948,Z 563.341,A 0.000,B 0.000,C 90.000,E1 97.352} C_DIS
LIN {X 0.176,Y -632.559,Z 563.335,A 0.000,B 0.000,C 90.000,E1 96.315} C_DIS
LIN {X 0.046,Y -635.072,Z 563.331,A 0.000,B 0.000,C 90.000,E1 95.568} C_DIS
LIN {X -0.263,Y -638.134,Z 563.325,A 0.000,B 0.000,C 90.000,E1 94.588} C_DIS
LIN {X 0.298,Y -640.173,Z 563.321,A 0.000,B 0.000,C 90.000,E1 93.784} C_DIS
LIN {X 0.241,Y -642.002,Z 563.317,A 0.000,B 0.000,C 90.000,E1 93.037} C_DIS
LIN {X -0.062,Y -643.982,Z 563.311,A 0.000,B 0.000,C 90.000,E1 92.064} C_DIS
LIN {X 0.142,Y -644.831,Z 563.309,A 0.000,B 0.000,C 90.000,E1 91.547} C_DIS
LIN {X -0.119,Y -646.204,Z 563.303,A 0.000,B 0.000,C 90.000,E1 90.573} C_DIS
LIN {X -0.138,Y -646.853,Z 563.299,A 0.000,B 0.000,C 90.000,E1 89.828} C_DIS
LIN {X 0.068,Y -647.135,Z 563.296,A 0.000,B 0.000,C 90.000,E1 89.312} C_DIS
LIN {X 0.054,Y -647.260,Z 563.292,A 0.000,B 0.000,C 90.000,E1 88.568} C_DIS
LIN {X 0.062,Y -647.155,Z 563.288,A 0.000,B 0.000,C 90.000,E1 87.822} C_DIS
LIN {X 0.043,Y -646.771,Z 563.284,A 0.000,B 0.000,C 90.000,E1 87.078} C_DIS
LIN {X 0.053,Y -646.181,Z 563.280,A 0.000,B 0.000,C 90.000,E1 86.331} C_DIS
LIN {X -0.174,Y -645.001,Z 563.274,A 0.000,B 0.000,C 90.000,E1 85.355} C_DIS
LIN {X 0.279,Y -643.548,Z 563.269,A 0.000,B 0.000,C 90.000,E1 84.318} C_DIS
LIN {X 0.078,Y -641.757,Z 563.263,A 0.000,B 0.000,C 90.000,E1 83.337} C_DIS
LIN {X 0.311,Y -638.858,Z 563.256,A 0.000,B 0.000,C 90.000,E1 82.064} C_DIS
LIN {X -0.137,Y -635.457,Z 563.249,A 0.000,B 0.000,C 90.000,E1 80.849} C_DIS
LIN {X 0.274,Y -632.468,Z 563.244,A 0.000,B 0.000,C 90.000,E1 79.803} C_DIS
LIN {X 0.019,Y -629.141,Z 563.238,A 0.000,B 0.000,C 90.000,E1 78.814} C_DIS
LIN {X 0.046,Y -626.458,Z 563.234,A 0.000,B 0.000,C 90.000,E1 78.049} C_DIS
LIN {X 0.050,Y -623.620,Z 563.229,A 0.000,B 0.000,C 90.000,E1 77.285} C_DIS
LIN {X 0.025,Y -620.441,Z 563.225,A 0.000,B 0.000,C 90.000,E1 76.520} C_DIS
LIN {X 0.192,Y -618.190,Z 563.222,A 0.000,B 0.000,C 90.000,E1 75.992} C_DIS
LIN {X 0.069,Y -613.956,Z 563.217,A 0.000,B 0.000,C 90.000,E1 75.102} C_DIS
LIN {X -0.005,Y -610.088,Z 563.213,A 0.000,B 0.000,C 90.000,E1 74.338} C_DIS
LIN {X -0.017,Y -605.852,Z 563.209,A 0.000,B 0.000,C 90.000,E1 73.559} C_DIS
LIN {X -0.119,Y -600.418,Z 563.204,A 0.000,B 0.000,C 90.000,E1 72.653} C_DIS
LIN {X -0.171,Y -596.185,Z 563.200,A 0.000,B 0.000,C 90.000,E1 72.000} C_DIS
LIN {X -0.076,Y -591.382,Z 563.196,A 0.000,B 0.000,C 90.000,E1 71.329} C_DIS
LIN {X -0.215,Y -586.158,Z 563.193,A 0.000,B 0.000,C 90.000,E1 70.678} C_DIS
LIN {X -0.208,Y -580.176,Z 563.189,A 0.000,B 0.000,C 90.000,E1 70.007} C_DIS
LIN {X 0.155,Y -576.488,Z 563.187,A 0.000,B 0.000,C 90.000,E1 69.571} C_DIS
LIN {X -0.169,Y -571.286,Z 563.184,A 0.000,B 0.000,C 90.000,E1 69.082} C_DIS
LIN {X -0.301,Y -567.161,Z 563.182,A 0.000,B 0.000,C 90.000,E1 68.720} C_DIS
LIN {X 0.157,Y -561.881,Z 563.179,A 0.000,B 0.000,C 90.000,E1 68.230} C_DIS
LIN {X 0.258,Y -556.474,Z 563.177,A 0.000,B 0.000,C 90.000,E1 67.794} C_DIS
LIN {X -0.217,Y -550.235,Z 563.174,A 0.000,B 0.000,C 90.000,E1 67.411} C_DIS
LIN {X 0.213,Y -543.736,Z 563.172,A 0.000,B 0.000,C 90.000,E1 66.975} C_DIS
LIN {X -0.111,Y -537.342,Z 563.170,A 0.000,B 0.000,C 90.000,E1 66.666} C_DIS
LIN {X 0.094,Y -530.523,Z 563.168,A 0.000,B 0.000,C 90.000,E1 66.305} C_DIS
LIN {X -0.001,Y -523.236,Z 563.167,A 0.000,B 0.000,C 90.000,E1 65.997} C_DIS
LIN {X -0.090,Y -516.320,Z 563.165,A 0.000,B 0.000,C 90.000,E1 65.717} C_DIS
LIN {X 0.013,Y -505.828,Z 563.163,A 0.000,B 0.000,C 90.000,E1 65.305} C_DIS
LIN {X -0.030,Y -484.706,Z 563.159,A 0.000,B 0.000,C 90.000,E1 64.537} C_DIS
LIN {X 0.076,Y -460.812,Z 563.153,A 0.000,B 0.000,C 90.000,E1 63.589} C_DIS
LIN {X -0.239,Y -458.226,Z 563.153,A 0.000,B 0.000,C 90.000,E1 63.512} C_DIS
LIN {X 0.136,Y -458.150,Z 563.153,A 0.000,B 0.000,C 90.000,E1 63.461} C_DIS
LIN {X 0.111,Y -455.398,Z 563.144,A 0.000,B 0.000,C 90.000,E1 61.847} C_DIS
LIN {X 0.026,Y -446.062,Z 563.120,A 0.000,B 0.000,C 90.000,E1 57.661} C_DIS
LIN {X -0.154,Y -444.287,Z 563.115,A 0.000,B 0.000,C 90.000,E1 56.707} C_DIS
LIN {X -0.096,Y -443.623,Z 563.113,A 0.000,B 0.000,C 90.000,E1 56.373} C_DIS
LIN {X -0.123,Y -438.752,Z 563.102,A 0.000,B 0.000,C 90.000,E1 54.402} C_DIS
LIN {X -0.163,Y -438.759,Z 563.102,A 0.000,B 0.000,C 90.000,E1 54.402} C_DIS
LIN {X -0.086,Y -442.129,Z 563.088,A 0.000,B 0.000,C 90.000,E1 51.778} C_DIS
LIN {X 0.163,Y -443.878,Z 563.080,A 0.000,B 0.000,C 90.000,E1 50.436} C_DIS
LIN {X -0.206,Y -445.939,Z 563.071,A 0.000,B 0.000,C 90.000,E1 48.852} C_DIS
LIN {X -0.242,Y -447.914,Z 563.062,A 0.000,B 0.000,C 90.000,E1 47.229} C_DIS
LIN {X 0.068,Y -449.427,Z 563.055,A 0.000,B 0.000,C 90.000,E1 45.891} C_DIS
LIN {X 0.074,Y -450.460,Z 563.050,A 0.000,B 0.000,C 90.000,E1 44.919} C_DIS
LIN {X 0.100,Y -451.585,Z 563.042,A 0.000,B 0.000,C 90.000,E1 43.623} C_DIS
LIN {X -0.174,Y -452.455,Z 563.035,A 0.000,B 0.000,C 90.000,E1 42.366} C_DIS
LIN {X -0.100,Y -453.047,Z 563.028,A 0.000,B 0.000,C 90.000,E1 41.067} C_DIS
LIN {X -0.019,Y -453.371,Z 563.021,A 0.000,B 0.000,C 90.000,E1 39.769} C_DIS
LIN {X 0.125,Y -453.520,Z 563.014,A 0.000,B 0.000,C 90.000,E1 38.463} C_DIS
LIN {X 0.276,Y -453.446,Z 563.007,A 0.000,B 0.000,C 90.000,E1 37.156} C_DIS
LIN {X -0.126,Y -453.208,Z 562.998,A 0.000,B 0.000,C 90.000,E1 35.598} C_DIS
LIN {X 0.268,Y -452.437,Z 562.985,A 0.000,B 0.000,C 90.000,E1 33.293} C_DIS
LIN {X 0.047,Y -451.955,Z 562.974,A 0.000,B 0.000,C 90.000,E1 31.386} C_DIS
LIN {X -0.038,Y -451.551,Z 562.964,A 0.000,B 0.000,C 90.000,E1 29.461} C_DIS
LIN {X -0.082,Y -451.014,Z 562.951,A 0.000,B 0.000,C 90.000,E1 27.206} C_DIS
LIN {X -0.211,Y -450.546,Z 562.940,A 0.000,B 0.000,C 90.000,E1 25.283} C_DIS
LIN {X 0.098,Y -450.377,Z 562.933,A 0.000,B 0.000,C 90.000,E1 23.951} C_DIS
LIN {X -0.018,Y -450.108,Z 562.922,A 0.000,B 0.000,C 90.000,E1 22.025} C_DIS
LIN {X -0.002,Y -449.989,Z 562.910,A 0.000,B 0.000,C 90.000,E1 19.758} C_DIS
LIN {X -0.148,Y -450.007,Z 562.897,A 0.000,B 0.000,C 90.000,E1 17.511} C_DIS
LIN {X -0.091,Y -450.386,Z 562.881,A 0.000,B 0.000,C 90.000,E1 14.592} C_DIS
LIN {X -0.101,Y -451.127,Z 562.867,A 0.000,B 0.000,C 90.000,E1 12.007} C_DIS
LIN {X -0.051,Y -452.468,Z 562.851,A 0.000,B 0.000,C 90.000,E1 9.095} C_DIS
LIN {X 0.201,Y -453.953,Z 562.836,A 0.000,B 0.000,C 90.000,E1 6.486} C_DIS
LIN {X 0.129,Y -455.652,Z 562.824,A 0.000,B 0.000,C 90.000,E1 4.245} C_DIS
LIN {X -0.102,Y -457.248,Z 562.813,A 0.000,B 0.000,C 90.000,E1 2.350} C_DIS
LIN {X -0.124,Y -459.496,Z 562.801,A 0.000,B 0.000,C 90.000,E1 0.115} C_DIS
LIN {X 0.057,Y -461.327,Z 562.792,A 0.000,B 0.000,C 90.000,E1 358.511} C_DIS
LIN {X 0.180,Y -463.343,Z 562.783,A 0.000,B 0.000,C 90.000,E1 356.906} C_DIS
LIN {X -0.093,Y -465.514,Z 562.774,A 0.000,B 0.000,C 90.000,E1 355.355} C_DIS
LIN {X -0.082,Y -467.356,Z 562.767,A 0.000,B 0.000,C 90.000,E1 354.090} C_DIS
LIN {X 0.011,Y -469.220,Z 562.760,A 0.000,B 0.000,C 90.000,E1 352.818} C_DIS
LIN {X -0.042,Y -471.445,Z 562.751,A 0.000,B 0.000,C 90.000,E1 351.254} C_DIS
LIN {X -0.057,Y -473.713,Z 562.743,A 0.000,B 0.000,C 90.000,E1 349.690} C_DIS
LIN {X 0.048,Y -476.151,Z 562.734,A 0.000,B 0.000,C 90.000,E1 348.117} C_DIS
LIN {X -0.079,Y -480.633,Z 562.719,A 0.000,B 0.000,C 90.000,E1 345.338} C_DIS
LIN {X 0.084,Y -485.063,Z 562.705,A 0.000,B 0.000,C 90.000,E1 342.851} C_DIS
LIN {X -0.144,Y -489.241,Z 562.693,A 0.000,B 0.000,C 90.000,E1 340.732} C_DIS
LIN {X -0.202,Y -491.610,Z 562.686,A 0.000,B 0.000,C 90.000,E1 339.518} C_DIS
LIN {X -0.007,Y -494.519,Z 562.678,A 0.000,B 0.000,C 90.000,E1 337.975} C_DIS
LIN {X -0.214,Y -497.368,Z 562.669,A 0.000,B 0.000,C 90.000,E1 336.485} C_DIS
LIN {X -0.168,Y -500.030,Z 562.661,A 0.000,B 0.000,C 90.000,E1 334.973} C_DIS
LIN {X -0.145,Y -502.087,Z 562.654,A 0.000,B 0.000,C 90.000,E1 333.768} C_DIS
LIN {X 0.207,Y -504.686,Z 562.646,A 0.000,B 0.000,C 90.000,E1 332.231} C_DIS
LIN {X -0.089,Y -508.123,Z 562.634,A 0.000,B 0.000,C 90.000,E1 330.177} C_DIS
LIN {X 0.049,Y -512.113,Z 562.621,A 0.000,B 0.000,C 90.000,E1 327.788} C_DIS
LIN {X 0.208,Y -514.641,Z 562.613,A 0.000,B 0.000,C 90.000,E1 326.294} C_DIS
LIN {X -0.023,Y -517.203,Z 562.605,A 0.000,B 0.000,C 90.000,E1 324.848} C_DIS
LIN {X 0.084,Y -519.850,Z 562.597,A 0.000,B 0.000,C 90.000,E1 323.371} C_DIS
LIN {X 0.003,Y -524.051,Z 562.584,A 0.000,B 0.000,C 90.000,E1 321.045} C_DIS
LIN {X 0.006,Y -528.185,Z 562.572,A 0.000,B 0.000,C 90.000,E1 319.013} C_DIS
LIN {X 0.054,Y -533.435,Z 562.560,A 0.000,B 0.000,C 90.000,E1 316.701} C_DIS
LIN {X 0.248,Y -538.264,Z 562.548,A 0.000,B 0.000,C 90.000,E1 314.676} C_DIS
LIN {X 0.219,Y -539.555,Z 562.545,A 0.000,B 0.000,C 90.000,E1 314.109} C_DIS
LIN {X 0.004,Y -543.188,Z 562.538,A 0.000,B 0.000,C 90.000,E1 312.852} C_DIS
LIN {X 0.225,Y -546.632,Z 562.533,A 0.000,B 0.000,C 90.000,E1 311.838} C_DIS
LIN {X -0.153,Y -548.142,Z 562.531,A 0.000,B 0.000,C 90.000,E1 311.595} C_DIS
LIN {X 0.198,Y -550.154,Z 562.529,A 0.000,B 0.000,C 90.000,E1 311.229} C_DIS
LIN {X 0.038,Y -551.431,Z 562.528,A 0.000,B 0.000,C 90.000,E1 311.105} C_DIS
LIN {X 0.175,Y -553.779,Z 562.527,A 0.000,B 0.000,C 90.000,E1 310.782} C_DIS
LIN {X -0.110,Y -556.926,Z 562.525,A 0.000,B 0.000,C 90.000,E1 310.458} C_DIS
LIN {X 0.342,Y -561.191,Z 562.523,A 0.000,B 0.000,C 90.000,E1 310.011} C_DIS
LIN {X 0.036,Y -566.639,Z 562.520,A 0.000,B 0.000,C 90.000,E1 309.600} C_DIS
LIN {X -0.112,Y -581.458,Z 562.514,A 0.000,B 0.000,C 90.000,E1 308.543} C_DIS
LIN {X 0.024,Y -589.871,Z 562.511,A 0.000,B 0.000,C 90.000,E1 307.890} C_DIS
LIN {X -0.001,Y -595.355,Z 562.508,A 0.000,B 0.000,C 90.000,E1 307.443} C_DIS
LIN {X -0.186,Y -601.949,Z 562.505,A 0.000,B 0.000,C 90.000,E1 306.870} C_DIS
LIN {X -0.195,Y -607.012,Z 562.502,A 0.000,B 0.000,C 90.000,E1 306.377} C_DIS
LIN {X 0.126,Y -610.668,Z 562.500,A 0.000,B 0.000,C 90.000,E1 305.964} C_DIS
LIN {X -0.370,Y -618.843,Z 562.495,A 0.000,B 0.000,C 90.000,E1 305.105} C_DIS
LIN {X -0.242,Y -626.587,Z 562.490,A 0.000,B 0.000,C 90.000,E1 304.199} C_DIS
LIN {X -0.025,Y -633.979,Z 562.485,A 0.000,B 0.000,C 90.000,E1 303.293} C_DIS
LIN {X -0.150,Y -638.753,Z 562.482,A 0.000,B 0.000,C 90.000,E1 302.673} C_DIS
LIN {X 0.278,Y -642.287,Z 562.479,A 0.000,B 0.000,C 90.000,E1 302.133} C_DIS
LIN {X -0.153,Y -645.459,Z 562.476,A 0.000,B 0.000,C 90.000,E1 301.671} C_DIS
LIN {X -0.192,Y -648.925,Z 562.472,A 0.000,B 0.000,C 90.000,E1 301.052} C_DIS
LIN {X 0.068,Y -652.459,Z 562.468,A 0.000,B 0.000,C 90.000,E1 300.285} C_DIS
LIN {X 0.131,Y -655.635,Z 562.464,A 0.000,B 0.000,C 90.000,E1 299.539} C_DIS
LIN {X -0.220,Y -657.620,Z 562.461,A 0.000,B 0.000,C 90.000,E1 299.077} C_DIS
LIN {X -0.044,Y -662.884,Z 562.453,A 0.000,B 0.000,C 90.000,E1 297.590} C_DIS
LIN {X -0.211,Y -665.582,Z 562.449,A 0.000,B 0.000,C 90.000,E1 296.873} C_DIS
LIN {X -0.063,Y -666.399,Z 562.448,A 0.000,B 0.000,C 90.000,E1 296.616} C_DIS
LIN {X 0.241,Y -667.648,Z 562.445,A 0.000,B 0.000,C 90.000,E1 296.104} C_DIS
LIN {X -0.205,Y -668.103,Z 562.444,A 0.000,B 0.000,C 90.000,E1 295.899} C_DIS
LIN {X -0.178,Y -667.730,Z 562.441,A 0.000,B 0.000,C 90.000,E1 295.412} C_DIS
LIN {X -0.020,Y -666.939,Z 562.440,A 0.000,B 0.000,C 90.000,E1 295.155} C_DIS
LIN {X 0.059,Y -666.332,Z 562.439,A 0.000,B 0.000,C 90.000,E1 295.027} C_DIS
LIN {X 0.212,Y -664.409,Z 562.438,A 0.000,B 0.000,C 90.000,E1 294.771} C_DIS
LIN {X 0.358,Y -662.796,Z 562.436,A 0.000,B 0.000,C 90.000,E1 294.515} C_DIS
LIN {X 0.429,Y -661.622,Z 562.436,A 0.000,B 0.000,C 90.000,E1 294.387} C_DIS
LIN {X 0.373,Y -655.188,Z 562.433,A 0.000,B 0.000,C 90.000,E1 293.951} C_DIS
LIN {X -0.163,Y -653.048,Z 562.433,A 0.000,B 0.000,C 90.000,E1 293.898} C_DIS
LIN {X 0.252,Y -646.496,Z 562.432,A 0.000,B 0.000,C 90.000,E1 293.643} C_DIS
LIN {X -0.185,Y -645.744,Z 562.431,A 0.000,B 0.000,C 90.000,E1 293.643} C_DIS
LIN {X -0.003,Y -640.768,Z 562.430,A 0.000,B 0.000,C 90.000,E1 293.462} C_DIS
LIN {X -0.276,Y -637.543,Z 562.430,A 0.000,B 0.000,C 90.000,E1 293.387} C_DIS
LIN {X 0.366,Y -623.603,Z 562.428,A 0.000,B 0.000,C 90.000,E1 292.950} C_DIS
LIN {X -0.251,Y -596.480,Z 562.423,A 0.000,B 0.000,C 90.000,E1 292.206} C_DIS
LIN {X 0.108,Y -581.019,Z 562.420,A 0.000,B 0.000,C 90.000,E1 291.663} C_DIS
LIN {X -0.264,Y -573.751,Z 562.419,A 0.000,B 0.000,C 90.000,E1 291.408} C_DIS
LIN {X -0.287,Y -568.443,Z 562.417,A 0.000,B 0.000,C 90.000,E1 291.099} C_DIS
LIN {X -0.269,Y -566.662,Z 562.416,A 0.000,B 0.000,C 90.000,E1 290.918} C_DIS
LIN {X -0.309,Y -566.638,Z 562.416,A 0.000,B 0.000,C 90.000,E1 290.918} C_DIS
LIN {X 0.076,Y -566.005,Z 562.415,A 0.000,B 0.000,C 90.000,E1 290.663} C_DIS
LIN {X -0.195,Y -565.743,Z 562.410,A 0.000,B 0.000,C 90.000,E1 289.885} C_DIS
LIN {X 0.016,Y -565.687,Z 562.403,A 0.000,B 0.000,C 90.000,E1 288.489} C_DIS
LIN {X -0.106,Y -565.484,Z 562.397,A 0.000,B 0.000,C 90.000,E1 287.402} C_DIS
LIN {X 0.081,Y -564.788,Z 562.388,A 0.000,B 0.000,C 90.000,E1 285.733} C_DIS
LIN {X 0.087,Y -564.059,Z 562.380,A 0.000,B 0.000,C 90.000,E1 284.356} C_DIS
LIN {X 0.241,Y -562.951,Z 562.369,A 0.000,B 0.000,C 90.000,E1 282.411} C_DIS
LIN {X -0.022,Y -561.964,Z 562.360,A 0.000,B 0.000,C 90.000,E1 280.782} C_DIS
LIN {X -0.142,Y -560.923,Z 562.349,A 0.000,B 0.000,C 90.000,E1 278.859} C_DIS
LIN {X 0.029,Y -560.230,Z 562.340,A 0.000,B 0.000,C 90.000,E1 277.182} C_DIS
LIN {X 0.119,Y -559.497,Z 562.331,A 0.000,B 0.000,C 90.000,E1 275.511} C_DIS
LIN {X 0.188,Y -558.857,Z 562.321,A 0.000,B 0.000,C 90.000,E1 273.841} C_DIS
LIN {X 0.253,Y -558.128,Z 562.311,A 0.000,B 0.000,C 90.000,E1 271.892} C_DIS
LIN {X 0.134,Y -557.551,Z 562.303,A 0.000,B 0.000,C 90.000,E1 270.516} C_DIS
LIN {X -0.006,Y -556.901,Z 562.295,A 0.000,B 0.000,C 90.000,E1 269.141} C_DIS
LIN {X 0.006,Y -555.897,Z 562.284,A 0.000,B 0.000,C 90.000,E1 267.192} C_DIS
LIN {X -0.227,Y -555.304,Z 562.278,A 0.000,B 0.000,C 90.000,E1 266.102} C_DIS
LIN {X 0.127,Y -554.653,Z 562.272,A 0.000,B 0.000,C 90.000,E1 264.951} C_DIS
LIN {X 0.094,Y -553.608,Z 562.263,A 0.000,B 0.000,C 90.000,E1 263.280} C_DIS
LIN {X -0.128,Y -552.854,Z 562.257,A 0.000,B 0.000,C 90.000,E1 262.186} C_DIS
LIN {X 0.141,Y -552.086,Z 562.252,A 0.000,B 0.000,C 90.000,E1 261.319} C_DIS
LIN {X 0.080,Y -550.571,Z 562.244,A 0.000,B 0.000,C 90.000,E1 259.926} C_DIS
LIN {X 0.202,Y -548.675,Z 562.235,A 0.000,B 0.000,C 90.000,E1 258.229} C_DIS
LIN {X 0.183,Y -547.260,Z 562.227,A 0.000,B 0.000,C 90.000,E1 256.825} C_DIS
LIN {X -0.179,Y -545.273,Z 562.218,A 0.000,B 0.000,C 90.000,E1 255.172} C_DIS
LIN {X 0.082,Y -543.149,Z 562.208,A 0.000,B 0.000,C 90.000,E1 253.449} C_DIS
LIN {X -0.071,Y -540.575,Z 562.199,A 0.000,B 0.000,C 90.000,E1 251.764} C_DIS
LIN {X -0.080,Y -539.205,Z 562.194,A 0.000,B 0.000,C 90.000,E1 250.913} C_DIS
LIN {X 0.147,Y -536.726,Z 562.186,A 0.000,B 0.000,C 90.000,E1 249.464} C_DIS
LIN {X 0.285,Y -535.097,Z 562.181,A 0.000,B 0.000,C 90.000,E1 248.592} C_DIS
LIN {X -0.082,Y -532.840,Z 562.175,A 0.000,B 0.000,C 90.000,E1 247.486} C_DIS
LIN {X -0.085,Y -529.723,Z 562.167,A 0.000,B 0.000,C 90.000,E1 246.049} C_DIS
LIN {X 0.245,Y -525.753,Z 562.157,A 0.000,B 0.000,C 90.000,E1 244.280} C_DIS
LIN {X -0.139,Y -522.168,Z 562.149,A 0.000,B 0.000,C 90.000,E1 242.871} C_DIS
LIN {X 0.113,Y -518.538,Z 562.141,A 0.000,B 0.000,C 90.000,E1 241.385} C_DIS
LIN {X 0.181,Y -515.474,Z 562.135,A 0.000,B 0.000,C 90.000,E1 240.205} C_DIS
LIN {X 0.107,Y -512.990,Z 562.130,A 0.000,B 0.000,C 90.000,E1 239.331} C_DIS
LIN {X -0.013,Y -508.525,Z 562.122,A 0.000,B 0.000,C 90.000,E1 237.867} C_DIS
LIN {X -0.174,Y -502.436,Z 562.110,A 0.000,B 0.000,C 90.000,E1 235.801} C_DIS
LIN {X 0.052,Y -498.196,Z 562.102,A 0.000,B 0.000,C 90.000,E1 234.276} C_DIS
LIN {X -0.197,Y -492.431,Z 562.090,A 0.000,B 0.000,C 90.000,E1 232.190} C_DIS
LIN {X -0.149,Y -485.999,Z 562.076,A 0.000,B 0.000,C 90.000,E1 229.747} C_DIS
LIN {X 0.078,Y -481.353,Z 562.066,A 0.000,B 0.000,C 90.000,E1 227.877} C_DIS
LIN {X 0.134,Y -474.379,Z 562.051,A 0.000,B 0.000,C 90.000,E1 225.081} C_DIS
LIN {X -0.047,Y -470.723,Z 562.042,A 0.000,B 0.000,C 90.000,E1 223.542} C_DIS
LIN {X -0.209,Y -466.329,Z 562.031,A 0.000,B 0.000,C 90.000,E1 221.676} C_DIS
LIN {X -0.171,Y -462.784,Z 562.023,A 0.000,B 0.000,C 90.000,E1 220.092} C_DIS
LIN {X -0.236,Y -460.031,Z 562.016,A 0.000,B 0.000,C 90.000,E1 218.830} C_DIS
LIN {X 0.121,Y -455.864,Z 562.005,A 0.000,B 0.000,C 90.000,E1 216.870} C_DIS
LIN {X 0.186,Y -451.165,Z 561.992,A 0.000,B 0.000,C 90.000,E1 214.612} C_DIS
LIN {X 0.237,Y -446.615,Z 561.980,A 0.000,B 0.000,C 90.000,E1 212.339} C_DIS
LIN {X 0.123,Y -444.111,Z 561.973,A 0.000,B 0.000,C 90.000,E1 211.052} C_DIS
LIN {X 0.224,Y -440.553,Z 561.962,A 0.000,B 0.000,C 90.000,E1 209.077} C_DIS
LIN {X 0.035,Y -437.129,Z 561.951,A 0.000,B 0.000,C 90.000,E1 207.129} C_DIS
LIN {X -0.041,Y -433.752,Z 561.940,A 0.000,B 0.000,C 90.000,E1 205.155} C_DIS
LIN {X 0.004,Y -430.003,Z 561.927,A 0.000,B 0.000,C 90.000,E1 202.823} C_DIS
LIN {X 0.201,Y -426.016,Z 561.912,A 0.000,B 0.000,C 90.000,E1 200.120} C_DIS
LIN {X -0.013,Y -422.390,Z 561.897,A 0.000,B 0.000,C 90.000,E1 197.457} C_DIS
LIN {X 0.027,Y -418.262,Z 561.878,A 0.000,B 0.000,C 90.000,E1 194.064} C_DIS
LIN {X -0.117,Y -416.886,Z 561.873,A 0.000,B 0.000,C 90.000,E1 193.063} C_DIS
LIN {X 0.153,Y -411.842,Z 561.852,A 0.000,B 0.000,C 90.000,E1 189.265} C_DIS
LIN {X -0.084,Y -408.053,Z 561.833,A 0.000,B 0.000,C 90.000,E1 185.853} C_DIS
LIN {X -0.137,Y -406.313,Z 561.823,A 0.000,B 0.000,C 90.000,E1 184.131} C_DIS
LIN {X 0.047,Y -403.245,Z 561.804,A 0.000,B 0.000,C 90.000,E1 180.630} C_DIS
LIN {X 0.169,Y -401.429,Z 561.788,A 0.000,B 0.000,C 90.000,E1 177.822} C_DIS
LIN {X -0.056,Y -400.445,Z 561.776,A 0.000,B 0.000,C 90.000,E1 175.755} C_DIS
LIN {X 0.104,Y -399.739,Z 561.763,A 0.000,B 0.000,C 90.000,E1 173.280} C_DIS
LIN {X -0.086,Y -399.417,Z 561.745,A 0.000,B 0.000,C 90.000,E1 170.151} C_DIS
LIN {X -0.140,Y -399.545,Z 561.730,A 0.000,B 0.000,C 90.000,E1 167.353} C_DIS
LIN {X 0.227,Y -400.358,Z 561.710,A 0.000,B 0.000,C 90.000,E1 163.795} C_DIS
LIN {X -0.089,Y -401.384,Z 561.695,A 0.000,B 0.000,C 90.000,E1 161.040} C_DIS
LIN {X 0.206,Y -402.338,Z 561.683,A 0.000,B 0.000,C 90.000,E1 158.901} C_DIS
LIN {X 0.018,Y -403.626,Z 561.669,A 0.000,B 0.000,C 90.000,E1 156.485} C_DIS
LIN {X -0.067,Y -404.813,Z 561.658,A 0.000,B 0.000,C 90.000,E1 154.409} C_DIS
LIN {X -0.053,Y -406.299,Z 561.644,A 0.000,B 0.000,C 90.000,E1 151.975} C_DIS
LIN {X -0.153,Y -407.222,Z 561.635,A 0.000,B 0.000,C 90.000,E1 150.255} C_DIS
LIN {X 0.245,Y -408.105,Z 561.623,A 0.000,B 0.000,C 90.000,E1 148.122} C_DIS
LIN {X 0.049,Y -408.716,Z 561.614,A 0.000,B 0.000,C 90.000,E1 146.421} C_DIS
LIN {X 0.089,Y -409.157,Z 561.604,A 0.000,B 0.000,C 90.000,E1 144.689} C_DIS
LIN {X -0.113,Y -409.450,Z 561.596,A 0.000,B 0.000,C 90.000,E1 143.336} C_DIS
LIN {X -0.156,Y -409.685,Z 561.587,A 0.000,B 0.000,C 90.000,E1 141.618} C_DIS
LIN {X 0.050,Y -409.822,Z 561.577,A 0.000,B 0.000,C 90.000,E1 139.865} C_DIS
LIN {X -0.103,Y -409.902,Z 561.568,A 0.000,B 0.000,C 90.000,E1 138.162} C_DIS
LIN {X 0.183,Y -410.000,Z 561.556,A 0.000,B 0.000,C 90.000,E1 136.053} C_DIS
LIN {X 0.030,Y -410.297,Z 561.543,A 0.000,B 0.000,C 90.000,E1 133.662} C_DIS
LIN {X 0.177,Y -410.484,Z 561.533,A 0.000,B 0.000,C 90.000,E1 131.919} C_DIS
LIN {X -0.065,Y -410.505,Z 561.522,A 0.000,B 0.000,C 90.000,E1 129.886} C_DIS
LIN {X 0.100,Y -410.326,Z 561.516,A 0.000,B 0.000,C 90.000,E1 128.830} C_DIS
LIN {X -0.148,Y -409.934,Z 561.510,A 0.000,B 0.000,C 90.000,E1 127.890} C_DIS
LIN {X -0.186,Y -409.940,Z 561.510,A 0.000,B 0.000,C 90.000,E1 127.890} C_DIS
LIN {X -0.003,Y -415.165,Z 561.501,A 0.000,B 0.000,C 90.000,E1 126.091} C_DIS
LIN {X 0.108,Y -416.847,Z 561.497,A 0.000,B 0.000,C 90.000,E1 125.391} C_DIS
LIN {X 0.037,Y -426.559,Z 561.476,A 0.000,B 0.000,C 90.000,E1 121.671} C_DIS
LIN {X 0.000,Y -430.623,Z 561.469,A 0.000,B 0.000,C 90.000,E1 120.335} C_DIS
LIN {X -0.048,Y -438.477,Z 561.451,A 0.000,B 0.000,C 90.000,E1 117.129} C_DIS
LIN {X -0.088,Y -438.517,Z 561.451,A 0.000,B 0.000,C 90.000,E1 117.129} C_DIS
LIN {X -0.188,Y -461.457,Z 561.445,A 0.000,B 0.000,C 90.000,E1 116.104} C_DIS
LIN {X -0.145,Y -482.147,Z 561.440,A 0.000,B 0.000,C 90.000,E1 115.155} C_DIS
LIN {X 0.046,Y -488.833,Z 561.438,A 0.000,B 0.000,C 90.000,E1 114.823} C_DIS
LIN {X 0.106,Y -502.203,Z 561.434,A 0.000,B 0.000,C 90.000,E1 114.155} C_DIS
LIN {X -0.027,Y -512.068,Z 561.431,A 0.000,B 0.000,C 90.000,E1 113.643} C_DIS
LIN {X -0.153,Y -523.369,Z 561.428,A 0.000,B 0.000,C 90.000,E1 113.025} C_DIS
LIN {X 0.202,Y -531.292,Z 561.425,A 0.000,B 0.000,C 90.000,E1 112.514} C_DIS
LIN {X 0.111,Y -539.142,Z 561.422,A 0.000,B 0.000,C 90.000,E1 112.025} C_DIS
LIN {X 0.327,Y -545.173,Z 561.420,A 0.000,B 0.000,C 90.000,E1 111.589} C_DIS
LIN {X 0.155,Y -551.168,Z 561.418,A 0.000,B 0.000,C 90.000,E1 111.173} C_DIS
LIN {X -0.060,Y -556.826,Z 561.415,A 0.000,B 0.000,C 90.000,E1 110.737} C_DIS
LIN {X -0.071,Y -562.235,Z 561.412,A 0.000,B 0.000,C 90.000,E1 110.248} C_DIS
LIN {X 0.138,Y -567.325,Z 561.410,A 0.000,B 0.000,C 90.000,E1 109.704} C_DIS
LIN {X 0.036,Y -573.139,Z 561.406,A 0.000,B 0.000,C 90.000,E1 109.033} C_DIS
LIN {X -0.060,Y -578.150,Z 561.402,A 0.000,B 0.000,C 90.000,E1 108.362} C_DIS
LIN {X 0.049,Y -580.785,Z 561.400,A 0.000,B 0.000,C 90.000,E1 107.946} C_DIS
LIN {X 0.211,Y -582.467,Z 561.398,A 0.000,B 0.000,C 90.000,E1 107.692} C_DIS
LIN {X 0.156,Y -587.228,Z 561.394,A 0.000,B 0.000,C 90.000,E1 106.913} C_DIS
LIN {X 0.000,Y -591.065,Z 561.390,A 0.000,B 0.000,C 90.000,E1 106.260} C_DIS
LIN {X -0.287,Y -595.925,Z 561.385,A 0.000,B 0.000,C 90.000,E1 105.371} C_DIS
LIN {X 0.281,Y -599.781,Z 561.381,A 0.000,B 0.000,C 90.000,E1 104.537} C_DIS
LIN {X 0.022,Y -603.432,Z 561.377,A 0.000,B 0.000,C 90.000,E1 103.772} C_DIS
LIN {X -0.136,Y -609.325,Z 561.369,A 0.000,B 0.000,C 90.000,E1 102.479} C_DIS
LIN {X -0.306,Y -612.620,Z 561.365,A 0.000,B 0.000,C 90.000,E1 101.715} C_DIS
LIN {X 0.155,Y -615.767,Z 561.361,A 0.000,B 0.000,C 90.000,E1 100.894} C_DIS
LIN {X 0.278,Y -617.740,Z 561.358,A 0.000,B 0.000,C 90.000,E1 100.366} C_DIS
LIN {X -0.028,Y -625.619,Z 561.346,A 0.000,B 0.000,C 90.000,E1 98.341} C_DIS
LIN {X -0.152,Y -628.545,Z 561.342,A 0.000,B 0.000,C 90.000,E1 97.587} C_DIS
LIN {X 0.090,Y -632.245,Z 561.336,A 0.000,B 0.000,C 90.000,E1 96.549} C_DIS
LIN {X -0.247,Y -635.699,Z 561.331,A 0.000,B 0.000,C 90.000,E1 95.568} C_DIS
LIN {X 0.087,Y -638.786,Z 561.325,A 0.000,B 0.000,C 90.000,E1 94.531} C_DIS
LIN {X -0.228,Y -641.502,Z 561.320,A 0.000,B 0.000,C 90.000,E1 93.555} C_DIS
LIN {X -0.272,Y -643.199,Z 561.315,A 0.000,B 0.000,C 90.000,E1 92.808} C_DIS
LIN {X 0.109,Y -645.147,Z 561.310,A 0.000,B 0.000,C 90.000,E1 91.776} C_DIS
LIN {X 0.074,Y -646.236,Z 561.306,A 0.000,B 0.000,C 90.000,E1 91.031} C_DIS
LIN {X 0.054,Y -647.160,Z 561.302,A 0.000,B 0.000,C 90.000,E1 90.286} C_DIS
LIN {X -0.175,Y -647.830,Z 561.296,A 0.000,B 0.000,C 90.000,E1 89.312} C_DIS
LIN {X -0.180,Y -647.919,Z 561.292,A 0.000,B 0.000,C 90.000,E1 88.568} C_DIS
LIN {X -0.167,Y -647.801,Z 561.288,A 0.000,B 0.000,C 90.000,E1 87.822} C_DIS
LIN {X 0.043,Y -647.594,Z 561.285,A 0.000,B 0.000,C 90.000,E1 87.306} C_DIS
LIN {X -0.163,Y -646.785,Z 561.280,A 0.000,B 0.000,C 90.000,E1 86.331} C_DIS
LIN {X 0.261,Y -645.562,Z 561.274,A 0.000,B 0.000,C 90.000,E1 85.298} C_DIS
LIN {X 0.080,Y -644.070,Z 561.268,A 0.000,B 0.000,C 90.000,E1 84.318} C_DIS
LIN {X 0.059,Y -642.712,Z 561.264,A 0.000,B 0.000,C 90.000,E1 83.571} C_DIS
LIN {X 0.273,Y -641.629,Z 561.262,A 0.000,B 0.000,C 90.000,E1 83.053} C_DIS
LIN {X 0.127,Y -639.235,Z 561.256,A 0.000,B 0.000,C 90.000,E1 82.064} C_DIS
LIN {X -0.135,Y -636.497,Z 561.250,A 0.000,B 0.000,C 90.000,E1 81.084} C_DIS
LIN {X 0.287,Y -633.469,Z 561.245,A 0.000,B 0.000,C 90.000,E1 80.038} C_DIS
LIN {X 0.042,Y -630.190,Z 561.239,A 0.000,B 0.000,C 90.000,E1 79.050} C_DIS
LIN {X 0.077,Y -627.482,Z 561.235,A 0.000,B 0.000,C 90.000,E1 78.285} C_DIS
LIN {X -0.115,Y -623.622,Z 561.229,A 0.000,B 0.000,C 90.000,E1 77.285} C_DIS
LIN {X 0.075,Y -621.538,Z 561.227,A 0.000,B 0.000,C 90.000,E1 76.756} C_DIS
LIN {X -0.158,Y -617.436,Z 561.221,A 0.000,B 0.000,C 90.000,E1 75.880} C_DIS
LIN {X -0.100,Y -613.687,Z 561.217,A 0.000,B 0.000,C 90.000,E1 75.102} C_DIS
LIN {X -0.151,Y -609.704,Z 561.213,A 0.000,B 0.000,C 90.000,E1 74.338} C_DIS
LIN {X -0.120,Y -606.124,Z 561.209,A 0.000,B 0.000,C 90.000,E1 73.685} C_DIS
LIN {X -0.134,Y -600.651,Z 561.204,A 0.000,B 0.000,C 90.000,E1 72.779} C_DIS
LIN {X 0.040,Y -595.549,Z 561.200,A 0.000,B 0.000,C 90.000,E1 72.000} C_DIS
LIN {X 0.248,Y -592.482,Z 561.198,A 0.000,B 0.000,C 90.000,E1 71.583} C_DIS
LIN {X -0.123,Y -589.463,Z 561.196,A 0.000,B 0.000,C 90.000,E1 71.221} C_DIS
LIN {X 0.241,Y -586.263,Z 561.193,A 0.000,B 0.000,C 90.000,E1 70.786} C_DIS
LIN {X -0.221,Y -580.428,Z 561.190,A 0.000,B 0.000,C 90.000,E1 70.188} C_DIS
LIN {X -0.135,Y -575.887,Z 561.187,A 0.000,B 0.000,C 90.000,E1 69.699} C_DIS
LIN {X -0.076,Y -571.001,Z 561.185,A 0.000,B 0.000,C 90.000,E1 69.209} C_DIS
LIN {X -0.131,Y -565.426,Z 561.182,A 0.000,B 0.000,C 90.000,E1 68.720} C_DIS
LIN {X -0.246,Y -559.771,Z 561.179,A 0.000,B 0.000,C 90.000,E1 68.284} C_DIS
LIN {X -0.014,Y -555.296,Z 561.177,A 0.000,B 0.000,C 90.000,E1 67.922} C_DIS
LIN {X 0.063,Y -548.808,Z 561.175,A 0.000,B 0.000,C 90.000,E1 67.486} C_DIS
LIN {X 0.180,Y -543.788,Z 561.173,A 0.000,B 0.000,C 90.000,E1 67.177} C_DIS
LIN {X 0.136,Y -535.213,Z 561.171,A 0.000,B 0.000,C 90.000,E1 66.741} C_DIS
LIN {X 0.218,Y -530.046,Z 561.170,A 0.000,B 0.000,C 90.000,E1 66.485} C_DIS
LIN {X 0.034,Y -519.581,Z 561.167,A 0.000,B 0.000,C 90.000,E1 66.049} C_DIS
LIN {X -0.310,Y -507.089,Z 561.164,A 0.000,B 0.000,C 90.000,E1 65.613} C_DIS
LIN {X 0.282,Y -487.731,Z 561.160,A 0.000,B 0.000,C 90.000,E1 64.845} C_DIS
LIN {X 0.169,Y -472.079,Z 561.157,A 0.000,B 0.000,C 90.000,E1 64.280} C_DIS
LIN {X -0.067,Y -458.704,Z 561.154,A 0.000,B 0.000,C 90.000,E1 63.768} C_DIS
LIN {X -0.102,Y -458.660,Z 561.154,A 0.000,B 0.000,C 90.000,E1 63.768} C_DIS
LIN {X -0.021,Y -455.676,Z 561.145,A 0.000,B 0.000,C 90.000,E1 62.025} C_DIS
LIN {X 0.084,Y -455.002,Z 561.143,A 0.000,B 0.000,C 90.000,E1 61.691} C_DIS
LIN {X 0.005,Y -445.760,Z 561.120,A 0.000,B 0.000,C 90.000,E1 57.502} C_DIS
LIN {X 0.197,Y -444.006,Z 561.114,A 0.000,B 0.000,C 90.000,E1 56.501} C_DIS
LIN {X -0.115,Y -439.126,Z 561.103,A 0.000,B 0.000,C 90.000,E1 54.562} C_DIS
LIN {X -0.155,Y -439.120,Z 561.103,A 0.000,B 0.000,C 90.000,E1 54.562} C_DIS
LIN {X -0.037,Y -441.262,Z 561.094,A 0.000,B 0.000,C 90.000,E1 52.924} C_DIS
LIN {X -0.087,Y -444.003,Z 561.083,A 0.000,B 0.000,C 90.000,E1 50.964} C_DIS
LIN {X 0.172,Y -446.133,Z 561.074,A 0.000,B 0.000,C 90.000,E1 49.299} C_DIS
LIN {X -0.165,Y -448.574,Z 561.063,A 0.000,B 0.000,C 90.000,E1 47.391} C_DIS
LIN {X 0.155,Y -450.085,Z 561.056,A 0.000,B 0.000,C 90.000,E1 46.053} C_DIS
LIN {X 0.177,Y -451.485,Z 561.049,A 0.000,B 0.000,C 90.000,E1 44.757} C_DIS
LIN {X 0.217,Y -452.571,Z 561.042,A 0.000,B 0.000,C 90.000,E1 43.461} C_DIS
LIN {X -0.042,Y -453.325,Z 561.034,A 0.000,B 0.000,C 90.000,E1 42.204} C_DIS
LIN {X 0.032,Y -453.781,Z 561.029,A 0.000,B 0.000,C 90.000,E1 41.229} C_DIS
LIN {X 0.127,Y -454.084,Z 561.022,A 0.000,B 0.000,C 90.000,E1 39.930} C_DIS
LIN {X 0.007,Y -454.226,Z 561.013,A 0.000,B 0.000,C 90.000,E1 38.338} C_DIS
LIN {X -0.188,Y -454.136,Z 561.006,A 0.000,B 0.000,C 90.000,E1 37.076} C_DIS
LIN {X 0.067,Y -453.921,Z 560.999,A 0.000,B 0.000,C 90.000,E1 35.758} C_DIS
LIN {X 0.049,Y -453.356,Z 560.990,A 0.000,B 0.000,C 90.000,E1 34.151} C_DIS
LIN {X 0.106,Y -452.784,Z 560.979,A 0.000,B 0.000,C 90.000,E1 32.212} C_DIS
LIN {X 0.050,Y -452.307,Z 560.968,A 0.000,B 0.000,C 90.000,E1 30.285} C_DIS
LIN {X 0.021,Y -451.983,Z 560.961,A 0.000,B 0.000,C 90.000,E1 28.999} C_DIS
LIN {X -0.013,Y -451.445,Z 560.949,A 0.000,B 0.000,C 90.000,E1 26.744} C_DIS
LIN {X 0.034,Y -450.878,Z 560.934,A 0.000,B 0.000,C 90.000,E1 24.155} C_DIS
LIN {X 0.110,Y -450.530,Z 560.923,A 0.000,B 0.000,C 90.000,E1 22.206} C_DIS
LIN {X 0.134,Y -450.373,Z 560.911,A 0.000,B 0.000,C 90.000,E1 19.939} C_DIS
LIN {X -0.001,Y -450.355,Z 560.898,A 0.000,B 0.000,C 90.000,E1 17.692} C_DIS
LIN {X -0.234,Y -450.579,Z 560.884,A 0.000,B 0.000,C 90.000,E1 15.134} C_DIS
LIN {X -0.126,Y -451.192,Z 560.870,A 0.000,B 0.000,C 90.000,E1 12.535} C_DIS
LIN {X -0.200,Y -452.269,Z 560.855,A 0.000,B 0.000,C 90.000,E1 9.962} C_DIS
LIN {X 0.076,Y -453.252,Z 560.844,A 0.000,B 0.000,C 90.000,E1 7.992} C_DIS
LIN {X 0.004,Y -455.177,Z 560.828,A 0.000,B 0.000,C 90.000,E1 5.106} C_DIS
LIN {X -0.034,Y -456.966,Z 560.816,A 0.000,B 0.000,C 90.000,E1 2.865} C_DIS
LIN {X 0.128,Y -459.442,Z 560.802,A 0.000,B 0.000,C 90.000,E1 0.286} C_DIS
LIN {X 0.059,Y -461.468,Z 560.792,A 0.000,B 0.000,C 90.000,E1 358.511} C_DIS
LIN {X 0.185,Y -463.469,Z 560.783,A 0.000,B 0.000,C 90.000,E1 356.906} C_DIS
LIN {X 0.164,Y -465.194,Z 560.776,A 0.000,B 0.000,C 90.000,E1 355.641} C_DIS
LIN {X -0.074,Y -467.466,Z 560.767,A 0.000,B 0.000,C 90.000,E1 354.090} C_DIS
LIN {X -0.167,Y -469.724,Z 560.758,A 0.000,B 0.000,C 90.000,E1 352.527} C_DIS
LIN {X -0.030,Y -471.507,Z 560.751,A 0.000,B 0.000,C 90.000,E1 351.254} C_DIS
LIN {X -0.044,Y -473.764,Z 560.743,A 0.000,B 0.000,C 90.000,E1 349.690} C_DIS
LIN {X 0.001,Y -476.683,Z 560.732,A 0.000,B 0.000,C 90.000,E1 347.813} C_DIS
LIN {X -0.064,Y -480.693,Z 560.719,A 0.000,B 0.000,C 90.000,E1 345.338} C_DIS
LIN {X 0.244,Y -484.540,Z 560.707,A 0.000,B 0.000,C 90.000,E1 343.142} C_DIS
LIN {X -0.126,Y -489.304,Z 560.693,A 0.000,B 0.000,C 90.000,E1 340.732} C_DIS
LIN {X -0.148,Y -492.257,Z 560.684,A 0.000,B 0.000,C 90.000,E1 339.209} C_DIS
LIN {X 0.060,Y -495.159,Z 560.676,A 0.000,B 0.000,C 90.000,E1 337.667} C_DIS
LIN {X -0.135,Y -497.979,Z 560.668,A 0.000,B 0.000,C 90.000,E1 336.177} C_DIS
LIN {X 0.199,Y -501.198,Z 560.658,A 0.000,B 0.000,C 90.000,E1 334.332} C_DIS
LIN {X 0.234,Y -504.793,Z 560.646,A 0.000,B 0.000,C 90.000,E1 332.231} C_DIS
LIN {X -0.312,Y -508.249,Z 560.634,A 0.000,B 0.000,C 90.000,E1 330.205} C_DIS
LIN {X 0.085,Y -512.276,Z 560.621,A 0.000,B 0.000,C 90.000,E1 327.788} C_DIS
LIN {X 0.246,Y -514.806,Z 560.613,A 0.000,B 0.000,C 90.000,E1 326.294} C_DIS
LIN {X 0.019,Y -517.382,Z 560.605,A 0.000,B 0.000,C 90.000,E1 324.848} C_DIS
LIN {X -0.288,Y -520.008,Z 560.597,A 0.000,B 0.000,C 90.000,E1 323.417} C_DIS
LIN {X 0.054,Y -524.220,Z 560.584,A 0.000,B 0.000,C 90.000,E1 321.045} C_DIS
LIN {X 0.061,Y -528.342,Z 560.572,A 0.000,B 0.000,C 90.000,E1 319.013} C_DIS
LIN {X 0.113,Y -533.597,Z 560.560,A 0.000,B 0.000,C 90.000,E1 316.701} C_DIS
LIN {X -0.070,Y -538.476,Z 560.548,A 0.000,B 0.000,C 90.000,E1 314.717} C_DIS
LIN {X 0.285,Y -539.742,Z 560.545,A 0.000,B 0.000,C 90.000,E1 314.109} C_DIS
LIN {X -0.119,Y -544.463,Z 560.536,A 0.000,B 0.000,C 90.000,E1 312.447} C_DIS
LIN {X -0.087,Y -547.243,Z 560.531,A 0.000,B 0.000,C 90.000,E1 311.595} C_DIS
LIN {X 0.188,Y -549.614,Z 560.529,A 0.000,B 0.000,C 90.000,E1 311.148} C_DIS
LIN {X 0.130,Y -550.515,Z 560.528,A 0.000,B 0.000,C 90.000,E1 310.943} C_DIS
LIN {X 0.074,Y -554.093,Z 560.525,A 0.000,B 0.000,C 90.000,E1 310.458} C_DIS
LIN {X 0.049,Y -557.918,Z 560.523,A 0.000,B 0.000,C 90.000,E1 310.048} C_DIS
LIN {X 0.015,Y -561.271,Z 560.521,A 0.000,B 0.000,C 90.000,E1 309.725} C_DIS
LIN {X -0.014,Y -565.601,Z 560.519,A 0.000,B 0.000,C 90.000,E1 309.358} C_DIS
LIN {X 0.201,Y -581.372,Z 560.512,A 0.000,B 0.000,C 90.000,E1 308.177} C_DIS
LIN {X 0.122,Y -589.950,Z 560.509,A 0.000,B 0.000,C 90.000,E1 307.523} C_DIS
LIN {X -0.008,Y -595.387,Z 560.506,A 0.000,B 0.000,C 90.000,E1 307.076} C_DIS
LIN {X 0.152,Y -600.578,Z 560.503,A 0.000,B 0.000,C 90.000,E1 306.583} C_DIS
LIN {X 0.064,Y -605.558,Z 560.501,A 0.000,B 0.000,C 90.000,E1 306.091} C_DIS
LIN {X 0.161,Y -611.646,Z 560.497,A 0.000,B 0.000,C 90.000,E1 305.438} C_DIS
LIN {X -0.114,Y -616.431,Z 560.494,A 0.000,B 0.000,C 90.000,E1 304.945} C_DIS
LIN {X -0.024,Y -625.367,Z 560.488,A 0.000,B 0.000,C 90.000,E1 303.913} C_DIS
LIN {X -0.210,Y -632.825,Z 560.484,A 0.000,B 0.000,C 90.000,E1 303.038} C_DIS
LIN {X 0.178,Y -636.747,Z 560.481,A 0.000,B 0.000,C 90.000,E1 302.498} C_DIS
LIN {X 0.077,Y -641.209,Z 560.477,A 0.000,B 0.000,C 90.000,E1 301.878} C_DIS
LIN {X -0.023,Y -644.429,Z 560.474,A 0.000,B 0.000,C 90.000,E1 301.386} C_DIS
LIN {X 0.153,Y -647.813,Z 560.471,A 0.000,B 0.000,C 90.000,E1 300.747} C_DIS
LIN {X 0.130,Y -650.772,Z 560.467,A 0.000,B 0.000,C 90.000,E1 300.129} C_DIS
LIN {X -0.153,Y -653.918,Z 560.463,A 0.000,B 0.000,C 90.000,E1 299.411} C_DIS
LIN {X 0.060,Y -655.925,Z 560.461,A 0.000,B 0.000,C 90.000,E1 298.899} C_DIS
LIN {X 0.034,Y -663.890,Z 560.448,A 0.000,B 0.000,C 90.000,E1 296.693} C_DIS
LIN {X -0.126,Y -665.708,Z 560.444,A 0.000,B 0.000,C 90.000,E1 295.976} C_DIS
LIN {X 0.172,Y -665.639,Z 560.442,A 0.000,B 0.000,C 90.000,E1 295.463} C_DIS
LIN {X 0.322,Y -665.246,Z 560.440,A 0.000,B 0.000,C 90.000,E1 295.207} C_DIS
LIN {X 0.113,Y -664.678,Z 560.440,A 0.000,B 0.000,C 90.000,E1 295.103} C_DIS
LIN {X -0.197,Y -661.457,Z 560.437,A 0.000,B 0.000,C 90.000,E1 294.643} C_DIS
LIN {X -0.127,Y -660.322,Z 560.436,A 0.000,B 0.000,C 90.000,E1 294.515} C_DIS
LIN {X -0.060,Y -658.853,Z 560.435,A 0.000,B 0.000,C 90.000,E1 294.387} C_DIS
LIN {X -0.269,Y -654.173,Z 560.434,A 0.000,B 0.000,C 90.000,E1 294.079} C_DIS
LIN {X 0.053,Y -652.252,Z 560.433,A 0.000,B 0.000,C 90.000,E1 293.951} C_DIS
LIN {X 0.281,Y -647.643,Z 560.432,A 0.000,B 0.000,C 90.000,E1 293.770} C_DIS
LIN {X 0.104,Y -644.894,Z 560.431,A 0.000,B 0.000,C 90.000,E1 293.643} C_DIS
LIN {X 0.036,Y -635.217,Z 560.430,A 0.000,B 0.000,C 90.000,E1 293.334} C_DIS
LIN {X -0.319,Y -600.034,Z 560.424,A 0.000,B 0.000,C 90.000,E1 292.333} C_DIS
LIN {X -0.280,Y -581.215,Z 560.421,A 0.000,B 0.000,C 90.000,E1 291.716} C_DIS
LIN {X -0.183,Y -573.922,Z 560.419,A 0.000,B 0.000,C 90.000,E1 291.408} C_DIS
LIN {X 0.259,Y -569.431,Z 560.417,A 0.000,B 0.000,C 90.000,E1 291.099} C_DIS
LIN {X 0.094,Y -567.098,Z 560.416,A 0.000,B 0.000,C 90.000,E1 290.865} C_DIS
LIN {X 0.053,Y -567.075,Z 560.416,A 0.000,B 0.000,C 90.000,E1 290.865} C_DIS
LIN {X 0.095,Y -566.490,Z 560.414,A 0.000,B 0.000,C 90.000,E1 290.556} C_DIS
LIN {X 0.001,Y -566.305,Z 560.409,A 0.000,B 0.000,C 90.000,E1 289.577} C_DIS
LIN {X 0.218,Y -566.213,Z 560.401,A 0.000,B 0.000,C 90.000,E1 288.181} C_DIS
LIN {X 0.100,Y -565.910,Z 560.395,A 0.000,B 0.000,C 90.000,E1 287.094} C_DIS
LIN {X -0.188,Y -565.491,Z 560.389,A 0.000,B 0.000,C 90.000,E1 286.024} C_DIS
LIN {X -0.011,Y -564.606,Z 560.380,A 0.000,B 0.000,C 90.000,E1 284.356} C_DIS
LIN {X 0.157,Y -563.502,Z 560.369,A 0.000,B 0.000,C 90.000,E1 282.411} C_DIS
LIN {X -0.094,Y -562.532,Z 560.360,A 0.000,B 0.000,C 90.000,E1 280.782} C_DIS
LIN {X 0.201,Y -561.643,Z 560.351,A 0.000,B 0.000,C 90.000,E1 279.095} C_DIS
LIN {X -0.091,Y -560.916,Z 560.341,A 0.000,B 0.000,C 90.000,E1 277.466} C_DIS
LIN {X 0.005,Y -560.200,Z 560.332,A 0.000,B 0.000,C 90.000,E1 275.796} C_DIS
LIN {X 0.043,Y -559.524,Z 560.323,A 0.000,B 0.000,C 90.000,E1 274.131} C_DIS
LIN {X 0.070,Y -558.869,Z 560.314,A 0.000,B 0.000,C 90.000,E1 272.465} C_DIS
LIN {X -0.036,Y -558.331,Z 560.306,A 0.000,B 0.000,C 90.000,E1 271.088} C_DIS
LIN {X -0.079,Y -557.553,Z 560.297,A 0.000,B 0.000,C 90.000,E1 269.427} C_DIS
LIN {X -0.047,Y -556.525,Z 560.286,A 0.000,B 0.000,C 90.000,E1 267.478} C_DIS
LIN {X -0.268,Y -555.932,Z 560.280,A 0.000,B 0.000,C 90.000,E1 266.388} C_DIS
LIN {X 0.164,Y -555.120,Z 560.272,A 0.000,B 0.000,C 90.000,E1 264.951} C_DIS
LIN {X 0.141,Y -554.043,Z 560.263,A 0.000,B 0.000,C 90.000,E1 263.280} C_DIS
LIN {X 0.044,Y -553.075,Z 560.255,A 0.000,B 0.000,C 90.000,E1 261.894} C_DIS
LIN {X -0.110,Y -551.961,Z 560.249,A 0.000,B 0.000,C 90.000,E1 260.792} C_DIS
LIN {X -0.281,Y -550.697,Z 560.243,A 0.000,B 0.000,C 90.000,E1 259.690} C_DIS
LIN {X -0.046,Y -548.472,Z 560.232,A 0.000,B 0.000,C 90.000,E1 257.701} C_DIS
LIN {X -0.168,Y -547.276,Z 560.225,A 0.000,B 0.000,C 90.000,E1 256.589} C_DIS
LIN {X -0.089,Y -545.635,Z 560.218,A 0.000,B 0.000,C 90.000,E1 255.172} C_DIS
LIN {X 0.021,Y -544.197,Z 560.211,A 0.000,B 0.000,C 90.000,E1 254.031} C_DIS
LIN {X -0.111,Y -543.016,Z 560.207,A 0.000,B 0.000,C 90.000,E1 253.196} C_DIS
LIN {X 0.259,Y -540.438,Z 560.197,A 0.000,B 0.000,C 90.000,E1 251.456} C_DIS
LIN {X 0.226,Y -537.519,Z 560.188,A 0.000,B 0.000,C 90.000,E1 249.752} C_DIS
LIN {X -0.102,Y -535.334,Z 560.181,A 0.000,B 0.000,C 90.000,E1 248.646} C_DIS
LIN {X -0.257,Y -532.426,Z 560.173,A 0.000,B 0.000,C 90.000,E1 247.230} C_DIS
LIN {X 0.033,Y -529.930,Z 560.167,A 0.000,B 0.000,C 90.000,E1 246.049} C_DIS
LIN {X 0.197,Y -526.602,Z 560.159,A 0.000,B 0.000,C 90.000,E1 244.588} C_DIS
LIN {X -0.089,Y -523.773,Z 560.153,A 0.000,B 0.000,C 90.000,E1 243.461} C_DIS
LIN {X -0.136,Y -519.373,Z 560.143,A 0.000,B 0.000,C 90.000,E1 241.719} C_DIS
LIN {X -0.059,Y -516.387,Z 560.136,A 0.000,B 0.000,C 90.000,E1 240.539} C_DIS
LIN {X 0.234,Y -513.108,Z 560.130,A 0.000,B 0.000,C 90.000,E1 239.331} C_DIS
LIN {X 0.016,Y -507.709,Z 560.120,A 0.000,B 0.000,C 90.000,E1 237.582} C_DIS
LIN {X -0.159,Y -501.640,Z 560.108,A 0.000,B 0.000,C 90.000,E1 235.515} C_DIS
LIN {X 0.180,Y -498.227,Z 560.102,A 0.000,B 0.000,C 90.000,E1 234.276} C_DIS
LIN {X -0.071,Y -492.457,Z 560.090,A 0.000,B 0.000,C 90.000,E1 232.190} C_DIS
LIN {X -0.023,Y -486.018,Z 560.076,A 0.000,B 0.000,C 90.000,E1 229.747} C_DIS
LIN {X -0.024,Y -480.557,Z 560.064,A 0.000,B 0.000,C 90.000,E1 227.595} C_DIS
LIN {X 0.257,Y -474.388,Z 560.051,A 0.000,B 0.000,C 90.000,E1 225.081} C_DIS
LIN {X 0.075,Y -470.718,Z 560.042,A 0.000,B 0.000,C 90.000,E1 223.542} C_DIS
LIN {X -0.087,Y -466.334,Z 560.032,A 0.000,B 0.000,C 90.000,E1 221.676} C_DIS
LIN {X -0.004,Y -462.075,Z 560.021,A 0.000,B 0.000,C 90.000,E1 219.769} C_DIS
LIN {X 0.013,Y -458.584,Z 560.012,A 0.000,B 0.000,C 90.000,E1 218.177} C_DIS
LIN {X -0.031,Y -455.155,Z 560.003,A 0.000,B 0.000,C 90.000,E1 216.583} C_DIS
LIN {X -0.069,Y -451.118,Z 559.993,A 0.000,B 0.000,C 90.000,E1 214.659} C_DIS
LIN {X -0.267,Y -446.564,Z 559.980,A 0.000,B 0.000,C 90.000,E1 212.418} C_DIS
LIN {X 0.005,Y -444.047,Z 559.973,A 0.000,B 0.000,C 90.000,E1 211.082} C_DIS
LIN {X -0.051,Y -440.488,Z 559.962,A 0.000,B 0.000,C 90.000,E1 209.127} C_DIS
LIN {X -0.030,Y -436.486,Z 559.949,A 0.000,B 0.000,C 90.000,E1 206.821} C_DIS
LIN {X 0.069,Y -433.145,Z 559.938,A 0.000,B 0.000,C 90.000,E1 204.823} C_DIS
LIN {X 0.125,Y -428.930,Z 559.923,A 0.000,B 0.000,C 90.000,E1 202.153} C_DIS
LIN {X 0.096,Y -425.482,Z 559.910,A 0.000,B 0.000,C 90.000,E1 199.812} C_DIS
LIN {X 0.084,Y -422.374,Z 559.897,A 0.000,B 0.000,C 90.000,E1 197.457} C_DIS
LIN {X 0.122,Y -418.252,Z 559.878,A 0.000,B 0.000,C 90.000,E1 194.064} C_DIS
LIN {X 0.032,Y -416.378,Z 559.871,A 0.000,B 0.000,C 90.000,E1 192.715} C_DIS
LIN {X -0.159,Y -411.857,Z 559.852,A 0.000,B 0.000,C 90.000,E1 189.321} C_DIS
LIN {X 0.010,Y -408.098,Z 559.833,A 0.000,B 0.000,C 90.000,E1 185.853} C_DIS
LIN {X -0.042,Y -406.388,Z 559.823,A 0.000,B 0.000,C 90.000,E1 184.131} C_DIS
LIN {X 0.144,Y -403.318,Z 559.804,A 0.000,B 0.000,C 90.000,E1 180.630} C_DIS
LIN {X -0.133,Y -401.527,Z 559.788,A 0.000,B 0.000,C 90.000,E1 177.879} C_DIS
LIN {X -0.024,Y -400.301,Z 559.773,A 0.000,B 0.000,C 90.000,E1 175.065} C_DIS
LIN {X 0.128,Y -399.704,Z 559.759,A 0.000,B 0.000,C 90.000,E1 172.591} C_DIS
LIN {X 0.023,Y -399.539,Z 559.745,A 0.000,B 0.000,C 90.000,E1 170.151} C_DIS
LIN {X -0.027,Y -399.667,Z 559.730,A 0.000,B 0.000,C 90.000,E1 167.353} C_DIS
LIN {X -0.121,Y -400.353,Z 559.712,A 0.000,B 0.000,C 90.000,E1 164.212} C_DIS
LIN {X -0.229,Y -401.070,Z 559.701,A 0.000,B 0.000,C 90.000,E1 162.127} C_DIS
LIN {X -0.079,Y -401.996,Z 559.689,A 0.000,B 0.000,C 90.000,E1 160.007} C_DIS
LIN {X 0.095,Y -403.193,Z 559.675,A 0.000,B 0.000,C 90.000,E1 157.539} C_DIS
LIN {X -0.163,Y -404.360,Z 559.664,A 0.000,B 0.000,C 90.000,E1 155.485} C_DIS
LIN {X -0.038,Y -405.173,Z 559.656,A 0.000,B 0.000,C 90.000,E1 154.076} C_DIS
LIN {X 0.087,Y -406.460,Z 559.644,A 0.000,B 0.000,C 90.000,E1 151.975} C_DIS
LIN {X -0.009,Y -407.409,Z 559.635,A 0.000,B 0.000,C 90.000,E1 150.255} C_DIS
LIN {X -0.082,Y -408.156,Z 559.625,A 0.000,B 0.000,C 90.000,E1 148.535} C_DIS
LIN {X 0.062,Y -408.806,Z 559.616,A 0.000,B 0.000,C 90.000,E1 146.786} C_DIS
LIN {X 0.098,Y -409.332,Z 559.606,A 0.000,B 0.000,C 90.000,E1 145.055} C_DIS
LIN {X 0.050,Y -409.700,Z 559.596,A 0.000,B 0.000,C 90.000,E1 143.336} C_DIS
LIN {X 0.011,Y -409.950,Z 559.587,A 0.000,B 0.000,C 90.000,E1 141.618} C_DIS
LIN {X -0.091,Y -410.086,Z 559.577,A 0.000,B 0.000,C 90.000,E1 139.908} C_DIS
LIN {X 0.074,Y -410.134,Z 559.568,A 0.000,B 0.000,C 90.000,E1 138.162} C_DIS
LIN {X -0.213,Y -410.225,Z 559.556,A 0.000,B 0.000,C 90.000,E1 136.134} C_DIS
LIN {X -0.077,Y -410.516,Z 559.543,A 0.000,B 0.000,C 90.000,E1 133.704} C_DIS
LIN {X -0.209,Y -410.694,Z 559.533,A 0.000,B 0.000,C 90.000,E1 132.000} C_DIS
LIN {X -0.028,Y -410.682,Z 559.524,A 0.000,B 0.000,C 90.000,E1 130.253} C_DIS
LIN {X -0.018,Y -410.501,Z 559.516,A 0.000,B 0.000,C 90.000,E1 128.874} C_DIS
LIN {X 0.014,Y -410.093,Z 559.510,A 0.000,B 0.000,C 90.000,E1 127.810} C_DIS
LIN {X -0.024,Y -410.102,Z 559.510,A 0.000,B 0.000,C 90.000,E1 127.810} C_DIS
LIN {X 0.205,Y -415.076,Z 559.501,A 0.000,B 0.000,C 90.000,E1 126.091} C_DIS
LIN {X -0.201,Y -416.003,Z 559.499,A 0.000,B 0.000,C 90.000,E1 125.804} C_DIS
LIN {X -0.095,Y -425.508,Z 559.478,A 0.000,B 0.000,C 90.000,E1 122.054} C_DIS
LIN {X 0.210,Y -430.535,Z 559.469,A 0.000,B 0.000,C 90.000,E1 120.335} C_DIS
LIN {X 0.063,Y -436.095,Z 559.456,A 0.000,B 0.000,C 90.000,E1 118.025} C_DIS
LIN {X 0.109,Y -439.255,Z 559.449,A 0.000,B 0.000,C 90.000,E1 116.821} C_DIS
LIN {X 0.070,Y -439.326,Z 559.449,A 0.000,B 0.000,C 90.000,E1 116.821} C_DIS
LIN {X -0.114,Y -462.576,Z 559.443,A 0.000,B 0.000,C 90.000,E1 115.796} C_DIS
LIN {X 0.027,Y -483.345,Z 559.438,A 0.000,B 0.000,C 90.000,E1 114.847} C_DIS
LIN {X 0.208,Y -490.040,Z 559.436,A 0.000,B 0.000,C 90.000,E1 114.515} C_DIS
LIN {X -0.261,Y -500.088,Z 559.434,A 0.000,B 0.000,C 90.000,E1 114.079} C_DIS
LIN {X -0.111,Y -511.587,Z 559.430,A 0.000,B 0.000,C 90.000,E1 113.462} C_DIS
LIN {X 0.001,Y -523.002,Z 559.427,A 0.000,B 0.000,C 90.000,E1 112.823} C_DIS
LIN {X -0.189,Y -532.557,Z 559.424,A 0.000,B 0.000,C 90.000,E1 112.280} C_DIS
LIN {X -0.033,Y -540.398,Z 559.421,A 0.000,B 0.000,C 90.000,E1 111.770} C_DIS
LIN {X -0.136,Y -547.592,Z 559.418,A 0.000,B 0.000,C 90.000,E1 111.280} C_DIS
LIN {X 0.031,Y -550.639,Z 559.417,A 0.000,B 0.000,C 90.000,E1 111.046} C_DIS
LIN {X -0.075,Y -556.323,Z 559.414,A 0.000,B 0.000,C 90.000,E1 110.610} C_DIS
LIN {X 0.089,Y -561.682,Z 559.412,A 0.000,B 0.000,C 90.000,E1 110.120} C_DIS
LIN {X 0.015,Y -566.677,Z 559.409,A 0.000,B 0.000,C 90.000,E1 109.631} C_DIS
LIN {X -0.025,Y -572.643,Z 559.405,A 0.000,B 0.000,C 90.000,E1 108.960} C_DIS
LIN {X -0.116,Y -577.827,Z 559.402,A 0.000,B 0.000,C 90.000,E1 108.290} C_DIS
LIN {X 0.196,Y -582.491,Z 559.398,A 0.000,B 0.000,C 90.000,E1 107.583} C_DIS
LIN {X 0.079,Y -587.422,Z 559.393,A 0.000,B 0.000,C 90.000,E1 106.804} C_DIS
LIN {X -0.146,Y -592.114,Z 559.389,A 0.000,B 0.000,C 90.000,E1 106.024} C_DIS
LIN {X 0.174,Y -597.040,Z 559.384,A 0.000,B 0.000,C 90.000,E1 105.064} C_DIS
LIN {X -0.048,Y -600.294,Z 559.380,A 0.000,B 0.000,C 90.000,E1 104.426} C_DIS
LIN {X -0.091,Y -603.431,Z 559.377,A 0.000,B 0.000,C 90.000,E1 103.772} C_DIS
LIN {X -0.248,Y -609.483,Z 559.369,A 0.000,B 0.000,C 90.000,E1 102.479} C_DIS
LIN {X 0.185,Y -612.837,Z 559.365,A 0.000,B 0.000,C 90.000,E1 101.658} C_DIS
LIN {X 0.048,Y -616.097,Z 559.361,A 0.000,B 0.000,C 90.000,E1 100.894} C_DIS
LIN {X 0.173,Y -618.094,Z 559.358,A 0.000,B 0.000,C 90.000,E1 100.366} C_DIS
LIN {X -0.124,Y -626.006,Z 559.346,A 0.000,B 0.000,C 90.000,E1 98.341} C_DIS
LIN {X -0.245,Y -628.963,Z 559.342,A 0.000,B 0.000,C 90.000,E1 97.587} C_DIS
LIN {X 0.003,Y -632.752,Z 559.336,A 0.000,B 0.000,C 90.000,E1 96.549} C_DIS
LIN {X -0.328,Y -636.250,Z 559.331,A 0.000,B 0.000,C 90.000,E1 95.568} C_DIS
LIN {X 0.013,Y -639.385,Z 559.325,A 0.000,B 0.000,C 90.000,E1 94.531} C_DIS
LIN {X -0.294,Y -642.132,Z 559.320,A 0.000,B 0.000,C 90.000,E1 93.555} C_DIS
LIN {X 0.311,Y -643.841,Z 559.315,A 0.000,B 0.000,C 90.000,E1 92.751} C_DIS
LIN {X 0.263,Y -645.339,Z 559.311,A 0.000,B 0.000,C 90.000,E1 92.007} C_DIS
LIN {X 0.251,Y -646.616,Z 559.307,A 0.000,B 0.000,C 90.000,E1 91.260} C_DIS
LIN {X 0.015,Y -647.845,Z 559.302,A 0.000,B 0.000,C 90.000,E1 90.286} C_DIS
LIN {X 0.012,Y -648.370,Z 559.297,A 0.000,B 0.000,C 90.000,E1 89.542} C_DIS
LIN {X 0.228,Y -648.605,Z 559.295,A 0.000,B 0.000,C 90.000,E1 89.026} C_DIS
LIN {X 0.032,Y -648.515,Z 559.289,A 0.000,B 0.000,C 90.000,E1 88.051} C_DIS
LIN {X 0.030,Y -648.247,Z 559.285,A 0.000,B 0.000,C 90.000,E1 87.306} C_DIS
LIN {X -0.167,Y -647.406,Z 559.280,A 0.000,B 0.000,C 90.000,E1 86.331} C_DIS
LIN {X 0.266,Y -646.149,Z 559.274,A 0.000,B 0.000,C 90.000,E1 85.298} C_DIS
LIN {X 0.092,Y -644.623,Z 559.269,A 0.000,B 0.000,C 90.000,E1 84.318} C_DIS
LIN {X 0.077,Y -643.238,Z 559.264,A 0.000,B 0.000,C 90.000,E1 83.571} C_DIS
LIN {X 0.295,Y -642.135,Z 559.262,A 0.000,B 0.000,C 90.000,E1 83.053} C_DIS
LIN {X 0.154,Y -639.660,Z 559.256,A 0.000,B 0.000,C 90.000,E1 82.064} C_DIS
LIN {X -0.284,Y -638.321,Z 559.253,A 0.000,B 0.000,C 90.000,E1 81.602} C_DIS
LIN {X 0.169,Y -635.313,Z 559.248,A 0.000,B 0.000,C 90.000,E1 80.557} C_DIS
LIN {X 0.141,Y -632.974,Z 559.243,A 0.000,B 0.000,C 90.000,E1 79.803} C_DIS
LIN {X 0.083,Y -630.401,Z 559.239,A 0.000,B 0.000,C 90.000,E1 79.050} C_DIS
LIN {X 0.315,Y -628.583,Z 559.236,A 0.000,B 0.000,C 90.000,E1 78.522} C_DIS
LIN {X -0.072,Y -623.615,Z 559.229,A 0.000,B 0.000,C 90.000,E1 77.285} C_DIS
LIN {X 0.118,Y -621.462,Z 559.227,A 0.000,B 0.000,C 90.000,E1 76.756} C_DIS
LIN {X -0.116,Y -617.300,Z 559.222,A 0.000,B 0.000,C 90.000,E1 75.880} C_DIS
LIN {X 0.038,Y -613.529,Z 559.217,A 0.000,B 0.000,C 90.000,E1 75.102} C_DIS
LIN {X 0.105,Y -610.119,Z 559.214,A 0.000,B 0.000,C 90.000,E1 74.448} C_DIS
LIN {X 0.140,Y -606.502,Z 559.210,A 0.000,B 0.000,C 90.000,E1 73.795} C_DIS
LIN {X 0.143,Y -602.514,Z 559.206,A 0.000,B 0.000,C 90.000,E1 73.142} C_DIS
LIN {X -0.183,Y -600.046,Z 559.204,A 0.000,B 0.000,C 90.000,E1 72.779} C_DIS
LIN {X 0.017,Y -595.674,Z 559.201,A 0.000,B 0.000,C 90.000,E1 72.127} C_DIS
LIN {X 0.227,Y -588.718,Z 559.196,A 0.000,B 0.000,C 90.000,E1 71.221} C_DIS
LIN {X -0.159,Y -585.317,Z 559.194,A 0.000,B 0.000,C 90.000,E1 70.859} C_DIS
LIN {X -0.051,Y -580.433,Z 559.191,A 0.000,B 0.000,C 90.000,E1 70.315} C_DIS
LIN {X -0.201,Y -577.675,Z 559.189,A 0.000,B 0.000,C 90.000,E1 70.061} C_DIS
LIN {X 0.048,Y -575.732,Z 559.188,A 0.000,B 0.000,C 90.000,E1 69.826} C_DIS
LIN {X 0.089,Y -570.695,Z 559.185,A 0.000,B 0.000,C 90.000,E1 69.337} C_DIS
LIN {X -0.212,Y -565.340,Z 559.183,A 0.000,B 0.000,C 90.000,E1 68.901} C_DIS
LIN {X -0.043,Y -559.215,Z 559.180,A 0.000,B 0.000,C 90.000,E1 68.411} C_DIS
LIN {X 0.131,Y -553.329,Z 559.178,A 0.000,B 0.000,C 90.000,E1 67.975} C_DIS
LIN {X 0.050,Y -548.379,Z 559.176,A 0.000,B 0.000,C 90.000,E1 67.667} C_DIS
LIN {X -0.089,Y -541.768,Z 559.174,A 0.000,B 0.000,C 90.000,E1 67.305} C_DIS
LIN {X 0.274,Y -534.838,Z 559.172,A 0.000,B 0.000,C 90.000,E1 66.922} C_DIS
LIN {X -0.101,Y -529.596,Z 559.171,A 0.000,B 0.000,C 90.000,E1 66.719} C_DIS
LIN {X 0.286,Y -519.177,Z 559.168,A 0.000,B 0.000,C 90.000,E1 66.230} C_DIS
LIN {X -0.140,Y -504.802,Z 559.165,A 0.000,B 0.000,C 90.000,E1 65.741} C_DIS
LIN {X -0.058,Y -487.123,Z 559.162,A 0.000,B 0.000,C 90.000,E1 65.101} C_DIS
LIN {X 0.031,Y -469.820,Z 559.158,A 0.000,B 0.000,C 90.000,E1 64.460} C_DIS
LIN {X 0.162,Y -459.249,Z 559.156,A 0.000,B 0.000,C 90.000,E1 64.024} C_DIS
LIN {X 0.129,Y -459.195,Z 559.156,A 0.000,B 0.000,C 90.000,E1 64.024} C_DIS
LIN {X -0.150,Y -455.650,Z 559.145,A 0.000,B 0.000,C 90.000,E1 62.025} C_DIS
LIN {X -0.159,Y -454.155,Z 559.141,A 0.000,B 0.000,C 90.000,E1 61.385} C_DIS
LIN {X -0.055,Y -445.129,Z 559.118,A 0.000,B 0.000,C 90.000,E1 57.168} C_DIS
LIN {X 0.068,Y -443.976,Z 559.114,A 0.000,B 0.000,C 90.000,E1 56.501} C_DIS
LIN {X 0.085,Y -439.483,Z 559.104,A 0.000,B 0.000,C 90.000,E1 54.689} C_DIS
LIN {X 0.045,Y -439.490,Z 559.104,A 0.000,B 0.000,C 90.000,E1 54.689} C_DIS
LIN {X 0.141,Y -442.437,Z 559.092,A 0.000,B 0.000,C 90.000,E1 52.557} C_DIS
LIN {X 0.088,Y -444.767,Z 559.083,A 0.000,B 0.000,C 90.000,E1 50.928} C_DIS
LIN {X 0.102,Y -446.523,Z 559.076,A 0.000,B 0.000,C 90.000,E1 49.622} C_DIS
LIN {X 0.071,Y -449.049,Z 559.065,A 0.000,B 0.000,C 90.000,E1 47.676} C_DIS
LIN {X 0.099,Y -450.956,Z 559.056,A 0.000,B 0.000,C 90.000,E1 46.053} C_DIS
LIN {X 0.133,Y -452.367,Z 559.049,A 0.000,B 0.000,C 90.000,E1 44.757} C_DIS
LIN {X 0.187,Y -453.402,Z 559.042,A 0.000,B 0.000,C 90.000,E1 43.461} C_DIS
LIN {X -0.060,Y -454.129,Z 559.034,A 0.000,B 0.000,C 90.000,E1 42.204} C_DIS
LIN {X 0.024,Y -454.558,Z 559.029,A 0.000,B 0.000,C 90.000,E1 41.229} C_DIS
LIN {X 0.131,Y -454.819,Z 559.022,A 0.000,B 0.000,C 90.000,E1 39.930} C_DIS
LIN {X 0.025,Y -454.940,Z 559.013,A 0.000,B 0.000,C 90.000,E1 38.338} C_DIS
LIN {X -0.160,Y -454.823,Z 559.006,A 0.000,B 0.000,C 90.000,E1 37.076} C_DIS
LIN {X 0.095,Y -454.525,Z 558.997,A 0.000,B 0.000,C 90.000,E1 35.438} C_DIS
LIN {X -0.018,Y -453.609,Z 558.983,A 0.000,B 0.000,C 90.000,E1 32.880} C_DIS
LIN {X 0.266,Y -452.966,Z 558.970,A 0.000,B 0.000,C 90.000,E1 30.590} C_DIS
LIN {X 0.112,Y -452.553,Z 558.961,A 0.000,B 0.000,C 90.000,E1 28.999} C_DIS
LIN {X 0.008,Y -452.019,Z 558.951,A 0.000,B 0.000,C 90.000,E1 27.078} C_DIS
LIN {X 0.056,Y -451.759,Z 558.945,A 0.000,B 0.000,C 90.000,E1 26.104} C_DIS
LIN {X -0.256,Y -451.328,Z 558.934,A 0.000,B 0.000,C 90.000,E1 24.207} C_DIS
LIN {X 0.242,Y -450.952,Z 558.924,A 0.000,B 0.000,C 90.000,E1 22.206} C_DIS
LIN {X -0.147,Y -450.750,Z 558.911,A 0.000,B 0.000,C 90.000,E1 19.993} C_DIS
LIN {X 0.151,Y -450.703,Z 558.898,A 0.000,B 0.000,C 90.000,E1 17.692} C_DIS
LIN {X 0.179,Y -450.866,Z 558.886,A 0.000,B 0.000,C 90.000,E1 15.426} C_DIS
LIN {X 0.046,Y -451.462,Z 558.870,A 0.000,B 0.000,C 90.000,E1 12.535} C_DIS
LIN {X -0.019,Y -452.498,Z 558.855,A 0.000,B 0.000,C 90.000,E1 9.962} C_DIS
LIN {X 0.023,Y -453.622,Z 558.843,A 0.000,B 0.000,C 90.000,E1 7.701} C_DIS
LIN {X -0.013,Y -455.111,Z 558.830,A 0.000,B 0.000,C 90.000,E1 5.454} C_DIS
LIN {X -0.042,Y -456.833,Z 558.818,A 0.000,B 0.000,C 90.000,E1 3.212} C_DIS
LIN {X 0.000,Y -459.908,Z 558.800,A 0.000,B 0.000,C 90.000,E1 360.000} C_DIS
LIN {X -0.195,Y -461.956,Z 558.790,A 0.000,B 0.000,C 90.000,E1 358.224} C_DIS
LIN {X -0.077,Y -464.877,Z 558.778,A 0.000,B 0.000,C 90.000,E1 355.988} C_DIS
LIN {X -0.065,Y -467.560,Z 558.767,A 0.000,B 0.000,C 90.000,E1 354.090} C_DIS
LIN {X -0.158,Y -469.786,Z 558.758,A 0.000,B 0.000,C 90.000,E1 352.527} C_DIS
LIN {X 0.195,Y -471.981,Z 558.750,A 0.000,B 0.000,C 90.000,E1 350.914} C_DIS
LIN {X -0.032,Y -473.794,Z 558.743,A 0.000,B 0.000,C 90.000,E1 349.690} C_DIS
LIN {X 0.013,Y -476.702,Z 558.732,A 0.000,B 0.000,C 90.000,E1 347.813} C_DIS
LIN {X -0.050,Y -480.754,Z 558.719,A 0.000,B 0.000,C 90.000,E1 345.338} C_DIS
LIN {X 0.118,Y -485.755,Z 558.703,A 0.000,B 0.000,C 90.000,E1 342.543} C_DIS
LIN {X -0.108,Y -489.369,Z 558.693,A 0.000,B 0.000,C 90.000,E1 340.732} C_DIS
LIN {X -0.130,Y -492.320,Z 558.684,A 0.000,B 0.000,C 90.000,E1 339.209} C_DIS
LIN {X 0.081,Y -495.222,Z 558.676,A 0.000,B 0.000,C 90.000,E1 337.667} C_DIS
LIN {X -0.114,Y -498.055,Z 558.668,A 0.000,B 0.000,C 90.000,E1 336.177} C_DIS
LIN {X 0.005,Y -501.291,Z 558.658,A 0.000,B 0.000,C 90.000,E1 334.357} C_DIS
LIN {X 0.189,Y -504.354,Z 558.648,A 0.000,B 0.000,C 90.000,E1 332.538} C_DIS
LIN {X -0.234,Y -507.362,Z 558.638,A 0.000,B 0.000,C 90.000,E1 330.795} C_DIS
LIN {X 0.005,Y -509.870,Z 558.629,A 0.000,B 0.000,C 90.000,E1 329.282} C_DIS
LIN {X 0.119,Y -512.427,Z 558.621,A 0.000,B 0.000,C 90.000,E1 327.788} C_DIS
LIN {X -0.146,Y -514.984,Z 558.613,A 0.000,B 0.000,C 90.000,E1 326.342} C_DIS
LIN {X 0.059,Y -517.577,Z 558.605,A 0.000,B 0.000,C 90.000,E1 324.848} C_DIS
LIN {X -0.243,Y -520.162,Z 558.597,A 0.000,B 0.000,C 90.000,E1 323.417} C_DIS
LIN {X -0.346,Y -524.975,Z 558.582,A 0.000,B 0.000,C 90.000,E1 320.803} C_DIS
LIN {X -0.052,Y -531.060,Z 558.566,A 0.000,B 0.000,C 90.000,E1 317.877} C_DIS
LIN {X -0.298,Y -535.833,Z 558.555,A 0.000,B 0.000,C 90.000,E1 315.891} C_DIS
LIN {X -0.018,Y -539.335,Z 558.547,A 0.000,B 0.000,C 90.000,E1 314.433} C_DIS
LIN {X 0.334,Y -543.701,Z 558.537,A 0.000,B 0.000,C 90.000,E1 312.690} C_DIS
LIN {X -0.016,Y -547.174,Z 558.531,A 0.000,B 0.000,C 90.000,E1 311.595} C_DIS
LIN {X 0.018,Y -547.980,Z 558.530,A 0.000,B 0.000,C 90.000,E1 311.310} C_DIS
LIN {X -0.157,Y -549.599,Z 558.527,A 0.000,B 0.000,C 90.000,E1 310.906} C_DIS
LIN {X 0.044,Y -550.596,Z 558.526,A 0.000,B 0.000,C 90.000,E1 310.744} C_DIS
LIN {X 0.094,Y -552.165,Z 558.525,A 0.000,B 0.000,C 90.000,E1 310.458} C_DIS
LIN {X 0.151,Y -554.497,Z 558.523,A 0.000,B 0.000,C 90.000,E1 310.172} C_DIS
LIN {X -0.209,Y -556.413,Z 558.522,A 0.000,B 0.000,C 90.000,E1 309.930} C_DIS
LIN {X -0.299,Y -558.282,Z 558.521,A 0.000,B 0.000,C 90.000,E1 309.725} C_DIS
LIN {X -0.163,Y -561.915,Z 558.519,A 0.000,B 0.000,C 90.000,E1 309.358} C_DIS
LIN {X -0.225,Y -566.351,Z 558.517,A 0.000,B 0.000,C 90.000,E1 308.991} C_DIS
LIN {X -0.062,Y -576.385,Z 558.512,A 0.000,B 0.000,C 90.000,E1 308.222} C_DIS
LIN {X -0.048,Y -583.561,Z 558.509,A 0.000,B 0.000,C 90.000,E1 307.684} C_DIS
LIN {X -0.046,Y -589.155,Z 558.507,A 0.000,B 0.000,C 90.000,E1 307.237} C_DIS
LIN {X 0.149,Y -593.294,Z 558.505,A 0.000,B 0.000,C 90.000,E1 306.870} C_DIS
LIN {X 0.265,Y -598.458,Z 558.502,A 0.000,B 0.000,C 90.000,E1 306.377} C_DIS
LIN {X -0.311,Y -604.654,Z 558.499,A 0.000,B 0.000,C 90.000,E1 305.804} C_DIS
LIN {X -0.246,Y -611.946,Z 558.495,A 0.000,B 0.000,C 90.000,E1 305.025} C_DIS
LIN {X 0.297,Y -618.983,Z 558.490,A 0.000,B 0.000,C 90.000,E1 304.199} C_DIS
LIN {X 0.055,Y -624.605,Z 558.487,A 0.000,B 0.000,C 90.000,E1 303.579} C_DIS
LIN {X -0.141,Y -631.104,Z 558.482,A 0.000,B 0.000,C 90.000,E1 302.832} C_DIS
LIN {X -0.275,Y -636.955,Z 558.478,A 0.000,B 0.000,C 90.000,E1 302.084} C_DIS
LIN {X 0.119,Y -639.641,Z 558.476,A 0.000,B 0.000,C 90.000,E1 301.671} C_DIS
LIN {X 0.007,Y -642.815,Z 558.473,A 0.000,B 0.000,C 90.000,E1 301.180} C_DIS
LIN {X 0.170,Y -646.346,Z 558.470,A 0.000,B 0.000,C 90.000,E1 300.541} C_DIS
LIN {X 0.131,Y -649.312,Z 558.466,A 0.000,B 0.000,C 90.000,E1 299.922} C_DIS
LIN {X -0.069,Y -653.349,Z 558.461,A 0.000,B 0.000,C 90.000,E1 298.949} C_DIS
LIN {X -0.094,Y -657.742,Z 558.454,A 0.000,B 0.000,C 90.000,E1 297.719} C_DIS
LIN {X -0.310,Y -660.545,Z 558.450,A 0.000,B 0.000,C 90.000,E1 297.001} C_DIS
LIN {X -0.048,Y -662.116,Z 558.447,A 0.000,B 0.000,C 90.000,E1 296.488} C_DIS
LIN {X 0.088,Y -662.799,Z 558.446,A 0.000,B 0.000,C 90.000,E1 296.232} C_DIS
LIN {X 0.227,Y -663.171,Z 558.444,A 0.000,B 0.000,C 90.000,E1 295.976} C_DIS
LIN {X -0.090,Y -663.254,Z 558.442,A 0.000,B 0.000,C 90.000,E1 295.515} C_DIS
LIN {X -0.234,Y -662.890,Z 558.440,A 0.000,B 0.000,C 90.000,E1 295.283} C_DIS
LIN {X -0.023,Y -660.529,Z 558.438,A 0.000,B 0.000,C 90.000,E1 294.899} C_DIS
LIN {X 0.045,Y -660.071,Z 558.438,A 0.000,B 0.000,C 90.000,E1 294.771} C_DIS
LIN {X 0.110,Y -659.247,Z 558.437,A 0.000,B 0.000,C 90.000,E1 294.643} C_DIS
LIN {X 0.105,Y -655.356,Z 558.435,A 0.000,B 0.000,C 90.000,E1 294.283} C_DIS
LIN {X -0.339,Y -653.846,Z 558.434,A 0.000,B 0.000,C 90.000,E1 294.207} C_DIS
LIN {X -0.185,Y -652.102,Z 558.434,A 0.000,B 0.000,C 90.000,E1 294.079} C_DIS
LIN {X 0.167,Y -649.738,Z 558.433,A 0.000,B 0.000,C 90.000,E1 293.951} C_DIS
LIN {X -0.067,Y -644.291,Z 558.432,A 0.000,B 0.000,C 90.000,E1 293.695} C_DIS
LIN {X 0.305,Y -640.092,Z 558.431,A 0.000,B 0.000,C 90.000,E1 293.515} C_DIS
LIN {X -0.271,Y -632.807,Z 558.430,A 0.000,B 0.000,C 90.000,E1 293.334} C_DIS
LIN {X -0.203,Y -610.064,Z 558.426,A 0.000,B 0.000,C 90.000,E1 292.642} C_DIS
LIN {X 0.073,Y -589.319,Z 558.422,A 0.000,B 0.000,C 90.000,E1 291.972} C_DIS
LIN {X -0.063,Y -579.549,Z 558.420,A 0.000,B 0.000,C 90.000,E1 291.642} C_DIS
LIN {X -0.139,Y -573.997,Z 558.419,A 0.000,B 0.000,C 90.000,E1 291.408} C_DIS
LIN {X 0.309,Y -569.639,Z 558.417,A 0.000,B 0.000,C 90.000,E1 291.099} C_DIS
LIN {X 0.280,Y -569.614,Z 558.417,A 0.000,B 0.000,C 90.000,E1 291.099} C_DIS
LIN {X 0.178,Y -567.733,Z 558.416,A 0.000,B 0.000,C 90.000,E1 290.865} C_DIS
LIN {X 0.135,Y -567.699,Z 558.416,A 0.000,B 0.000,C 90.000,E1 290.865} C_DIS
LIN {X 0.053,Y -567.053,Z 558.414,A 0.000,B 0.000,C 90.000,E1 290.556} C_DIS
LIN {X 0.249,Y -566.776,Z 558.404,A 0.000,B 0.000,C 90.000,E1 288.725} C_DIS
LIN {X 0.141,Y -566.638,Z 558.398,A 0.000,B 0.000,C 90.000,E1 287.638} C_DIS
LIN {X -0.196,Y -566.059,Z 558.389,A 0.000,B 0.000,C 90.000,E1 286.024} C_DIS
LIN {X -0.006,Y -565.158,Z 558.380,A 0.000,B 0.000,C 90.000,E1 284.356} C_DIS
LIN {X 0.176,Y -564.058,Z 558.369,A 0.000,B 0.000,C 90.000,E1 282.411} C_DIS
LIN {X 0.098,Y -562.995,Z 558.358,A 0.000,B 0.000,C 90.000,E1 280.489} C_DIS
LIN {X 0.150,Y -561.840,Z 558.346,A 0.000,B 0.000,C 90.000,E1 278.276} C_DIS
LIN {X -0.292,Y -561.109,Z 558.337,A 0.000,B 0.000,C 90.000,E1 276.663} C_DIS
LIN {X 0.072,Y -560.767,Z 558.332,A 0.000,B 0.000,C 90.000,E1 275.796} C_DIS
LIN {X 0.036,Y -560.209,Z 558.325,A 0.000,B 0.000,C 90.000,E1 274.416} C_DIS
LIN {X -0.016,Y -559.653,Z 558.317,A 0.000,B 0.000,C 90.000,E1 273.037} C_DIS
LIN {X 0.064,Y -558.868,Z 558.306,A 0.000,B 0.000,C 90.000,E1 271.088} C_DIS
LIN {X -0.053,Y -558.209,Z 558.298,A 0.000,B 0.000,C 90.000,E1 269.714} C_DIS
LIN {X -0.003,Y -557.173,Z 558.288,A 0.000,B 0.000,C 90.000,E1 267.764} C_DIS
LIN {X -0.137,Y -556.406,Z 558.280,A 0.000,B 0.000,C 90.000,E1 266.388} C_DIS
LIN {X -0.183,Y -555.415,Z 558.271,A 0.000,B 0.000,C 90.000,E1 264.723} C_DIS
LIN {X -0.206,Y -554.303,Z 558.261,A 0.000,B 0.000,C 90.000,E1 263.053} C_DIS
LIN {X -0.226,Y -553.309,Z 558.254,A 0.000,B 0.000,C 90.000,E1 261.659} C_DIS
LIN {X 0.197,Y -551.834,Z 558.246,A 0.000,B 0.000,C 90.000,E1 260.218} C_DIS
LIN {X 0.025,Y -549.202,Z 558.233,A 0.000,B 0.000,C 90.000,E1 257.993} C_DIS
LIN {X 0.017,Y -547.676,Z 558.226,A 0.000,B 0.000,C 90.000,E1 256.589} C_DIS
LIN {X 0.102,Y -546.010,Z 558.218,A 0.000,B 0.000,C 90.000,E1 255.172} C_DIS
LIN {X 0.067,Y -544.574,Z 558.211,A 0.000,B 0.000,C 90.000,E1 254.047} C_DIS
LIN {X -0.124,Y -542.479,Z 558.204,A 0.000,B 0.000,C 90.000,E1 252.653} C_DIS
LIN {X -0.048,Y -540.726,Z 558.197,A 0.000,B 0.000,C 90.000,E1 251.511} C_DIS
LIN {X -0.068,Y -537.806,Z 558.188,A 0.000,B 0.000,C 90.000,E1 249.806} C_DIS
LIN {X 0.112,Y -535.593,Z 558.181,A 0.000,B 0.000,C 90.000,E1 248.646} C_DIS
LIN {X -0.040,Y -532.659,Z 558.174,A 0.000,B 0.000,C 90.000,E1 247.230} C_DIS
LIN {X 0.253,Y -530.160,Z 558.167,A 0.000,B 0.000,C 90.000,E1 246.049} C_DIS
LIN {X -0.282,Y -526.813,Z 558.159,A 0.000,B 0.000,C 90.000,E1 244.665} C_DIS
LIN {X 0.058,Y -523.222,Z 558.151,A 0.000,B 0.000,C 90.000,E1 243.179} C_DIS
LIN {X 0.010,Y -518.776,Z 558.141,A 0.000,B 0.000,C 90.000,E1 241.435} C_DIS
LIN {X 0.086,Y -515.727,Z 558.135,A 0.000,B 0.000,C 90.000,E1 240.255} C_DIS
LIN {X -0.242,Y -513.261,Z 558.130,A 0.000,B 0.000,C 90.000,E1 239.410} C_DIS
LIN {X 0.244,Y -507.833,Z 558.120,A 0.000,B 0.000,C 90.000,E1 237.582} C_DIS
LIN {X 0.069,Y -501.738,Z 558.109,A 0.000,B 0.000,C 90.000,E1 235.515} C_DIS
LIN {X 0.004,Y -498.305,Z 558.102,A 0.000,B 0.000,C 90.000,E1 234.322} C_DIS
LIN {X 0.156,Y -492.526,Z 558.090,A 0.000,B 0.000,C 90.000,E1 232.190} C_DIS
LIN {X 0.204,Y -486.085,Z 558.077,A 0.000,B 0.000,C 90.000,E1 229.747} C_DIS
LIN {X -0.122,Y -480.599,Z 558.065,A 0.000,B 0.000,C 90.000,E1 227.634} C_DIS
LIN {X -0.190,Y -474.430,Z 558.051,A 0.000,B 0.000,C 90.000,E1 225.162} C_DIS
LIN {X -0.026,Y -470.756,Z 558.042,A 0.000,B 0.000,C 90.000,E1 223.581} C_DIS
LIN {X 0.134,Y -466.367,Z 558.032,A 0.000,B 0.000,C 90.000,E1 221.676} C_DIS
LIN {X -0.079,Y -462.076,Z 558.021,A 0.000,B 0.000,C 90.000,E1 219.806} C_DIS
LIN {X 0.232,Y -458.593,Z 558.012,A 0.000,B 0.000,C 90.000,E1 218.177} C_DIS
LIN {X 0.187,Y -455.152,Z 558.003,A 0.000,B 0.000,C 90.000,E1 216.583} C_DIS
LIN {X -0.111,Y -451.114,Z 557.993,A 0.000,B 0.000,C 90.000,E1 214.692} C_DIS
LIN {X -0.054,Y -446.555,Z 557.980,A 0.000,B 0.000,C 90.000,E1 212.418} C_DIS
LIN {X 0.063,Y -441.650,Z 557.966,A 0.000,B 0.000,C 90.000,E1 209.795} C_DIS
LIN {X -0.041,Y -436.989,Z 557.951,A 0.000,B 0.000,C 90.000,E1 207.180} C_DIS
LIN {X -0.133,Y -434.202,Z 557.942,A 0.000,B 0.000,C 90.000,E1 205.540} C_DIS
LIN {X -0.096,Y -431.482,Z 557.933,A 0.000,B 0.000,C 90.000,E1 203.875} C_DIS
LIN {X 0.134,Y -428.393,Z 557.922,A 0.000,B 0.000,C 90.000,E1 201.844} C_DIS
LIN {X -0.260,Y -424.550,Z 557.907,A 0.000,B 0.000,C 90.000,E1 199.214} C_DIS
LIN {X 0.058,Y -421.921,Z 557.895,A 0.000,B 0.000,C 90.000,E1 197.149} C_DIS
LIN {X -0.089,Y -418.241,Z 557.878,A 0.000,B 0.000,C 90.000,E1 194.120} C_DIS
LIN {X -0.181,Y -416.409,Z 557.871,A 0.000,B 0.000,C 90.000,E1 192.771} C_DIS
LIN {X 0.069,Y -411.500,Z 557.850,A 0.000,B 0.000,C 90.000,E1 188.973} C_DIS
LIN {X 0.203,Y -408.156,Z 557.833,A 0.000,B 0.000,C 90.000,E1 185.853} C_DIS
LIN {X 0.152,Y -406.478,Z 557.823,A 0.000,B 0.000,C 90.000,E1 184.131} C_DIS
LIN {X -0.064,Y -403.402,Z 557.804,A 0.000,B 0.000,C 90.000,E1 180.688} C_DIS
LIN {X 0.064,Y -401.638,Z 557.788,A 0.000,B 0.000,C 90.000,E1 177.879} C_DIS
LIN {X 0.177,Y -400.432,Z 557.773,A 0.000,B 0.000,C 90.000,E1 175.065} C_DIS
LIN {X -0.110,Y -399.702,Z 557.753,A 0.000,B 0.000,C 90.000,E1 171.602} C_DIS
LIN {X 0.201,Y -399.637,Z 557.742,A 0.000,B 0.000,C 90.000,E1 169.454} C_DIS
LIN {X -0.206,Y -399.788,Z 557.730,A 0.000,B 0.000,C 90.000,E1 167.409} C_DIS
LIN {X -0.067,Y -400.270,Z 557.716,A 0.000,B 0.000,C 90.000,E1 164.936} C_DIS
LIN {X -0.063,Y -400.919,Z 557.705,A 0.000,B 0.000,C 90.000,E1 162.834} C_DIS
LIN {X 0.054,Y -401.979,Z 557.691,A 0.000,B 0.000,C 90.000,E1 160.369} C_DIS
LIN {X 0.080,Y -403.157,Z 557.677,A 0.000,B 0.000,C 90.000,E1 157.922} C_DIS
LIN {X -0.019,Y -404.306,Z 557.666,A 0.000,B 0.000,C 90.000,E1 155.845} C_DIS
LIN {X -0.064,Y -405.136,Z 557.658,A 0.000,B 0.000,C 90.000,E1 154.460} C_DIS
LIN {X -0.202,Y -406.177,Z 557.648,A 0.000,B 0.000,C 90.000,E1 152.743} C_DIS
LIN {X 0.143,Y -407.007,Z 557.641,A 0.000,B 0.000,C 90.000,E1 151.307} C_DIS
LIN {X -0.055,Y -407.742,Z 557.633,A 0.000,B 0.000,C 90.000,E1 149.950} C_DIS
LIN {X 0.081,Y -408.523,Z 557.623,A 0.000,B 0.000,C 90.000,E1 148.201} C_DIS
LIN {X -0.110,Y -409.126,Z 557.614,A 0.000,B 0.000,C 90.000,E1 146.501} C_DIS
LIN {X 0.018,Y -409.586,Z 557.606,A 0.000,B 0.000,C 90.000,E1 145.102} C_DIS
LIN {X -0.105,Y -410.011,Z 557.595,A 0.000,B 0.000,C 90.000,E1 143.050} C_DIS
LIN {X -0.139,Y -410.241,Z 557.585,A 0.000,B 0.000,C 90.000,E1 141.331} C_DIS
LIN {X 0.027,Y -410.344,Z 557.576,A 0.000,B 0.000,C 90.000,E1 139.585} C_DIS
LIN {X -0.221,Y -410.398,Z 557.564,A 0.000,B 0.000,C 90.000,E1 137.553} C_DIS
LIN {X -0.223,Y -410.502,Z 557.553,A 0.000,B 0.000,C 90.000,E1 135.486} C_DIS
LIN {X 0.066,Y -410.767,Z 557.541,A 0.000,B 0.000,C 90.000,E1 133.380} C_DIS
LIN {X 0.085,Y -410.906,Z 557.533,A 0.000,B 0.000,C 90.000,E1 132.000} C_DIS
LIN {X 0.108,Y -410.873,Z 557.526,A 0.000,B 0.000,C 90.000,E1 130.620} C_DIS
LIN {X 0.017,Y -410.789,Z 557.520,A 0.000,B 0.000,C 90.000,E1 129.600} C_DIS
LIN {X 0.187,Y -410.571,Z 557.514,A 0.000,B 0.000,C 90.000,E1 128.543} C_DIS
LIN {X 0.198,Y -410.254,Z 557.510,A 0.000,B 0.000,C 90.000,E1 127.729} C_DIS
LIN {X 0.161,Y -410.255,Z 557.510,A 0.000,B 0.000,C 90.000,E1 127.729} C_DIS
LIN {X -0.070,Y -414.946,Z 557.501,A 0.000,B 0.000,C 90.000,E1 126.171} C_DIS
LIN {X 0.104,Y -415.908,Z 557.499,A 0.000,B 0.000,C 90.000,E1 125.804} C_DIS
LIN {X -0.014,Y -425.390,Z 557.478,A 0.000,B 0.000,C 90.000,E1 122.084} C_DIS
LIN {X -0.071,Y -430.407,Z 557.469,A 0.000,B 0.000,C 90.000,E1 120.413} C_DIS
LIN {X -0.066,Y -432.009,Z 557.465,A 0.000,B 0.000,C 90.000,E1 119.745} C_DIS
LIN {X 0.094,Y -440.040,Z 557.448,A 0.000,B 0.000,C 90.000,E1 116.539} C_DIS
LIN {X 0.055,Y -440.087,Z 557.448,A 0.000,B 0.000,C 90.000,E1 116.539} C_DIS
LIN {X -0.042,Y -465.411,Z 557.441,A 0.000,B 0.000,C 90.000,E1 115.412} C_DIS
LIN {X -0.039,Y -484.422,Z 557.437,A 0.000,B 0.000,C 90.000,E1 114.567} C_DIS
LIN {X -0.082,Y -491.249,Z 557.435,A 0.000,B 0.000,C 90.000,E1 114.259} C_DIS
LIN {X -0.041,Y -501.259,Z 557.432,A 0.000,B 0.000,C 90.000,E1 113.770} C_DIS
LIN {X 0.130,Y -512.807,Z 557.429,A 0.000,B 0.000,C 90.000,E1 113.153} C_DIS
LIN {X -0.057,Y -522.632,Z 557.426,A 0.000,B 0.000,C 90.000,E1 112.642} C_DIS
LIN {X 0.192,Y -530.615,Z 557.423,A 0.000,B 0.000,C 90.000,E1 112.153} C_DIS
LIN {X 0.095,Y -533.887,Z 557.422,A 0.000,B 0.000,C 90.000,E1 111.972} C_DIS
LIN {X 0.045,Y -540.124,Z 557.420,A 0.000,B 0.000,C 90.000,E1 111.589} C_DIS
LIN {X 0.070,Y -547.277,Z 557.417,A 0.000,B 0.000,C 90.000,E1 111.099} C_DIS
LIN {X -0.215,Y -550.300,Z 557.416,A 0.000,B 0.000,C 90.000,E1 110.918} C_DIS
LIN {X 0.164,Y -556.168,Z 557.414,A 0.000,B 0.000,C 90.000,E1 110.429} C_DIS
